LIN {X 0,Y 569.385,Z 629.743,A -85,B 0,C 180,E1 27677.459,E2 27677.459} C_VEL
LIN {X 0,Y 569.347,Z 629.746,A -85,B 0,C 180,E1 27674.085,E2 27674.085} C_VEL
LIN {X 0,Y 569.375,Z 629.741,A -85,B 0,C 180,E1 27670.786,E2 27670.786} C_VEL
LIN {X 0,Y 569.404,Z 629.994,A -85,B 0,C 180,E1 27669.564,E2 27669.564} C_VEL
LIN {X 0,Y 577.566,Z 654.883,A -85,B 0,C 180,E1 27666.47,E2 27666.47} C_VEL
LIN {X 0,Y 582.986,Z 672.69,A -85,B 0,C 180,E1 27664.382,E2 27664.382} C_VEL
LIN {X 0,Y 582.582,Z 679.276,A -85,B 0,C 180,E1 27663.798,E2 27663.798} C_VEL
LIN {X 0,Y 590.179,Z 717.868,A -85,B 0,C 180,E1 27662.715,E2 27662.715} C_VEL
LIN {X 0,Y 584.592,Z 960.2,A -85,B 0,C 180,E1 27659.286,E2 27659.286} C_VEL
LIN {X 0,Y 583.754,Z 989.804,A -85,B 0,C 180,E1 27658.818,E2 27658.818} C_VEL
LIN {X 0,Y 582.732,Z 1011.571,A -85,B 0,C 180,E1 27658.307,E2 27658.307} C_VEL
LIN {X 0,Y 581.47,Z 1033.5,A -85,B 0,C 180,E1 27657.607,E2 27657.607} C_VEL
LIN {X 0,Y 580.045,Z 1054.405,A -85,B 0,C 180,E1 27656.753,E2 27656.753} C_VEL
LIN {X 0,Y 578.394,Z 1076.21,A -85,B 0,C 180,E1 27655.657,E2 27655.657} C_VEL
LIN {X 0,Y 576.83,Z 1095.761,A -85,B 0,C 180,E1 27654.473,E2 27654.473} C_VEL
LIN {X 0,Y 575.231,Z 1114.452,A -85,B 0,C 180,E1 27653.13,E2 27653.13} C_VEL
LIN {X 0,Y 573.746,Z 1131.579,A -85,B 0,C 180,E1 27651.681,E2 27651.681} C_VEL
LIN {X 0,Y 572.318,Z 1148.38,A -85,B 0,C 180,E1 27650.023,E2 27650.023} C_VEL
LIN {X 0,Y 571.147,Z 1162.85,A -85,B 0,C 180,E1 27648.366,E2 27648.366} C_VEL
LIN {X 0,Y 570.1,Z 1176.631,A -85,B 0,C 180,E1 27646.505,E2 27646.505} C_VEL
LIN {X 0,Y 569.274,Z 1188.963,A -85,B 0,C 180,E1 27644.545,E2 27644.545} C_VEL
LIN {X 0,Y 568.7,Z 1199.347,A -85,B 0,C 180,E1 27642.591,E2 27642.591} C_VEL
LIN {X 0,Y 568.31,Z 1208.283,A -85,B 0,C 180,E1 27640.542,E2 27640.542} C_VEL
LIN {X 0,Y 568.098,Z 1215.604,A -85,B 0,C 180,E1 27638.439,E2 27638.439} C_VEL
LIN {X 0,Y 567.982,Z 1221.411,A -85,B 0,C 180,E1 27636.265,E2 27636.265} C_VEL
LIN {X 0,Y 567.957,Z 1225.194,A -85,B 0,C 180,E1 27634.239,E2 27634.239} C_VEL
LIN {X 0,Y 567.958,Z 1227.62,A -85,B 0,C 180,E1 27632.016,E2 27632.016} C_VEL
LIN {X 0,Y 567.959,Z 1228.354,A -85,B 0,C 180,E1 27629.898,E2 27629.898} C_VEL
LIN {X 0,Y 567.961,Z 1227.38,A -85,B 0,C 180,E1 27627.779,E2 27627.779} C_VEL
LIN {X 0,Y 567.963,Z 1224.652,A -85,B 0,C 180,E1 27625.556,E2 27625.556} C_VEL
LIN {X 0,Y 567.992,Z 1220.397,A -85,B 0,C 180,E1 27623.428,E2 27623.428} C_VEL
LIN {X 0,Y 568.113,Z 1214.604,A -85,B 0,C 180,E1 27621.395,E2 27621.395} C_VEL
LIN {X 0,Y 568.343,Z 1206.72,A -85,B 0,C 180,E1 27619.251,E2 27619.251} C_VEL
LIN {X 0,Y 568.733,Z 1197.343,A -85,B 0,C 180,E1 27617.2,E2 27617.2} C_VEL
LIN {X 0,Y 569.298,Z 1186.437,A -85,B 0,C 180,E1 27615.245,E2 27615.245} C_VEL
LIN {X 0,Y 570.048,Z 1174.137,A -85,B 0,C 180,E1 27613.386,E2 27613.386} C_VEL
LIN {X 0,Y 570.986,Z 1160.553,A -85,B 0,C 180,E1 27611.625,E2 27611.625} C_VEL
LIN {X 0,Y 572.146,Z 1144.814,A -85,B 0,C 180,E1 27609.89,E2 27609.89} C_VEL
LIN {X 0,Y 573.396,Z 1128.474,A -85,B 0,C 180,E1 27608.351,E2 27608.351} C_VEL
LIN {X 0,Y 574.818,Z 1109.922,A -85,B 0,C 180,E1 27606.85,E2 27606.85} C_VEL
LIN {X 0,Y 576.284,Z 1091.145,A -85,B 0,C 180,E1 27605.554,E2 27605.554} C_VEL
LIN {X 0,Y 577.77,Z 1070.527,A -85,B 0,C 180,E1 27604.363,E2 27604.363} C_VEL
LIN {X 0,Y 579.158,Z 1050.131,A -85,B 0,C 180,E1 27603.383,E2 27603.383} C_VEL
LIN {X 0,Y 580.584,Z 1027.426,A -85,B 0,C 180,E1 27602.493,E2 27602.493} C_VEL
LIN {X 0,Y 581.823,Z 1005.201,A -85,B 0,C 180,E1 27601.811,E2 27601.811} C_VEL
LIN {X 0,Y 582.893,Z 981.742,A -85,B 0,C 180,E1 27601.283,E2 27601.283} C_VEL
LIN {X 0,Y 586.569,Z 850.583,A -85,B 0,C 180,E1 27599.246,E2 27599.246} C_VEL
LIN {X 0,Y 590.83,Z 750.197,A -85,B 0,C 180,E1 27597.537,E2 27597.537} C_VEL
LIN {X 0,Y 592.379,Z 716.599,A -85,B 0,C 180,E1 27596.915,E2 27596.915} C_VEL
LIN {X 0,Y 588.657,Z 690.874,A -85,B 0,C 180,E1 27595.977,E2 27595.977} C_VEL
LIN {X 0,Y 585.547,Z 674.638,A -85,B 0,C 180,E1 27595.245,E2 27595.245} C_VEL
LIN {X 0,Y 583.11,Z 669.092,A -85,B 0,C 180,E1 27594.818,E2 27594.818} C_VEL
LIN {X 0,Y 580.106,Z 657.836,A -85,B 0,C 180,E1 27593.11,E2 27593.11} C_VEL
LIN {X 0,Y 577.035,Z 648.434,A -85,B 0,C 180,E1 27591.4,E2 27591.4} C_VEL
LIN {X 0,Y 574.123,Z 641.138,A -85,B 0,C 180,E1 27589.715,E2 27589.715} C_VEL
LIN {X 0,Y 572.591,Z 637.429,A -85,B 0,C 180,E1 27588.669,E2 27588.669} C_VEL
LIN {X 0,Y 570.972,Z 633.671,A -85,B 0,C 180,E1 27587.334,E2 27587.334} C_VEL
LIN {X 0,Y 569.377,Z 629.969,A -85,B 0,C 180,E1 27585.337,E2 27585.337} C_VEL
LIN {X 0,Y 569.384,Z 629.746,A -85,B 0,C 180,E1 27582.176,E2 27582.176} C_VEL
LIN {X 0,Y 569.39,Z 630.021,A -85,B 0,C 180,E1 27580.923,E2 27580.923} C_VEL
LIN {X 0,Y 571.02,Z 633.725,A -85,B 0,C 180,E1 27578.81,E2 27578.81} C_VEL
LIN {X 0,Y 573.022,Z 638.744,A -85,B 0,C 180,E1 27577.015,E2 27577.015} C_VEL
LIN {X 0,Y 574.473,Z 642.072,A -85,B 0,C 180,E1 27576.094,E2 27576.094} C_VEL
LIN {X 0,Y 579.186,Z 648.73,A -85,B 0,C 180,E1 27575.256,E2 27575.256} C_VEL
LIN {X 0,Y 583.805,Z 655.292,A -85,B 0,C 180,E1 27574.531,E2 27574.531} C_VEL
LIN {X 0,Y 590.369,Z 666.287,A -85,B 0,C 180,E1 27573.561,E2 27573.561} C_VEL
LIN {X 0,Y 594.016,Z 673.562,A -85,B 0,C 180,E1 27573.045,E2 27573.045} C_VEL
LIN {X 0,Y 588.975,Z 770.536,A -85,B 0,C 180,E1 27571.31,E2 27571.31} C_VEL
LIN {X 0,Y 585.467,Z 865.563,A -85,B 0,C 180,E1 27569.75,E2 27569.75} C_VEL
LIN {X 0,Y 583.506,Z 937.323,A -85,B 0,C 180,E1 27568.629,E2 27568.629} C_VEL
LIN {X 0,Y 582.639,Z 960.337,A -85,B 0,C 180,E1 27568.084,E2 27568.084} C_VEL
LIN {X 0,Y 581.532,Z 982.034,A -85,B 0,C 180,E1 27567.385,E2 27567.385} C_VEL
LIN {X 0,Y 580.245,Z 1003.436,A -85,B 0,C 180,E1 27566.509,E2 27566.509} C_VEL
LIN {X 0,Y 578.839,Z 1023.952,A -85,B 0,C 180,E1 27565.477,E2 27565.477} C_VEL
LIN {X 0,Y 577.353,Z 1043.592,A -85,B 0,C 180,E1 27564.289,E2 27564.289} C_VEL
LIN {X 0,Y 575.82,Z 1062.116,A -85,B 0,C 180,E1 27562.946,E2 27562.946} C_VEL
LIN {X 0,Y 574.347,Z 1079.125,A -85,B 0,C 180,E1 27561.495,E2 27561.495} C_VEL
LIN {X 0,Y 572.947,Z 1095.168,A -85,B 0,C 180,E1 27559.897,E2 27559.897} C_VEL
LIN {X 0,Y 571.741,Z 1109.387,A -85,B 0,C 180,E1 27558.245,E2 27558.245} C_VEL
LIN {X 0,Y 570.667,Z 1122.187,A -85,B 0,C 180,E1 27556.492,E2 27556.492} C_VEL
LIN {X 0,Y 569.736,Z 1134.33,A -85,B 0,C 180,E1 27554.537,E2 27554.537} C_VEL
LIN {X 0,Y 569.076,Z 1144.509,A -85,B 0,C 180,E1 27552.586,E2 27552.586} C_VEL
LIN {X 0,Y 568.574,Z 1153.183,A -85,B 0,C 180,E1 27550.54,E2 27550.54} C_VEL
LIN {X 0,Y 568.254,Z 1160.43,A -85,B 0,C 180,E1 27548.4,E2 27548.4} C_VEL
LIN {X 0,Y 568.086,Z 1165.74,A -85,B 0,C 180,E1 27546.368,E2 27546.368} C_VEL
LIN {X 0,Y 567.995,Z 1169.579,A -85,B 0,C 180,E1 27544.242,E2 27544.242} C_VEL
LIN {X 0,Y 567.96,Z 1171.94,A -85,B 0,C 180,E1 27542.02,E2 27542.02} C_VEL
LIN {X 0,Y 567.963,Z 1172.683,A -85,B 0,C 180,E1 27539.901,E2 27539.901} C_VEL
LIN {X 0,Y 567.956,Z 1171.775,A -85,B 0,C 180,E1 27537.783,E2 27537.783} C_VEL
LIN {X 0,Y 567.991,Z 1169.228,A -85,B 0,C 180,E1 27535.56,E2 27535.56} C_VEL
LIN {X 0,Y 568.078,Z 1165.231,A -85,B 0,C 180,E1 27533.433,E2 27533.433} C_VEL
LIN {X 0,Y 568.246,Z 1159.452,A -85,B 0,C 180,E1 27531.299,E2 27531.299} C_VEL
LIN {X 0,Y 568.575,Z 1151.939,A -85,B 0,C 180,E1 27529.157,E2 27529.157} C_VEL
LIN {X 0,Y 569.088,Z 1143.026,A -85,B 0,C 180,E1 27527.109,E2 27527.109} C_VEL
LIN {X 0,Y 569.782,Z 1132.656,A -85,B 0,C 180,E1 27525.157,E2 27525.157} C_VEL
LIN {X 0,Y 570.734,Z 1120.273,A -85,B 0,C 180,E1 27523.2,E2 27523.2} C_VEL
LIN {X 0,Y 571.903,Z 1106.402,A -85,B 0,C 180,E1 27521.343,E2 27521.343} C_VEL
LIN {X 0,Y 573.241,Z 1091.506,A -85,B 0,C 180,E1 27519.639,E2 27519.639} C_VEL
LIN {X 0,Y 574.707,Z 1074.964,A -85,B 0,C 180,E1 27518.036,E2 27518.036} C_VEL
LIN {X 0,Y 576.258,Z 1057.5,A -85,B 0,C 180,E1 27516.59,E2 27516.59} C_VEL
LIN {X 0,Y 577.834,Z 1039.197,A -85,B 0,C 180,E1 27515.295,E2 27515.295} C_VEL
LIN {X 0,Y 579.41,Z 1019.369,A -85,B 0,C 180,E1 27514.116,E2 27514.116} C_VEL
LIN {X 0,Y 580.837,Z 999.457,A -85,B 0,C 180,E1 27513.138,E2 27513.138} C_VEL
LIN {X 0,Y 582.221,Z 977.603,A -85,B 0,C 180,E1 27512.266,E2 27512.266} C_VEL
LIN {X 0,Y 583.325,Z 956.104,A -85,B 0,C 180,E1 27511.593,E2 27511.593} C_VEL
LIN {X 0,Y 584.219,Z 933.964,A -85,B 0,C 180,E1 27511.089,E2 27511.089} C_VEL
LIN {X 0,Y 585.088,Z 897.354,A -85,B 0,C 180,E1 27510.542,E2 27510.542} C_VEL
LIN {X 0,Y 590.004,Z 687.581,A -85,B 0,C 180,E1 27507.575,E2 27507.575} C_VEL
LIN {X 0,Y 590.303,Z 670.134,A -85,B 0,C 180,E1 27507.312,E2 27507.312} C_VEL
LIN {X 0,Y 576.833,Z 644.025,A -85,B 0,C 180,E1 27506.064,E2 27506.064} C_VEL
LIN {X 0,Y 569.547,Z 630.919,A -85,B 0,C 180,E1 27505.383,E2 27505.383} C_VEL
LIN {X 0,Y 569.316,Z 629.751,A -85,B 0,C 180,E1 27505.32,E2 27505.32} C_VEL
LIN {X 0,Y 569.345,Z 629.744,A -85,B 0,C 180,E1 27501.948,E2 27501.948} C_VEL
LIN {X 0,Y 569.377,Z 629.741,A -85,B 0,C 180,E1 27498.732,E2 27498.732} C_VEL
LIN {X 0,Y 569.363,Z 629.745,A -85,B 0,C 180,E1 27496.965,E2 27496.965} C_VEL
LIN {X 0,Y 568.378,Z 629.865,A -85,B 0,C 180,E1 27496.19,E2 27496.19} C_VEL
LIN {X 0,Y 561.876,Z 630.685,A -85,B 0,C 180,E1 27493.958,E2 27493.958} C_VEL
LIN {X 0,Y 561.411,Z 630.738,A -85,B 0,C 180,E1 27493.448,E2 27493.448} C_VEL
LIN {X 0,Y 561.412,Z 630.736,A -85,B 0,C 180,E1 27490.28,E2 27490.28} C_VEL
LIN {X 0,Y 561.376,Z 630.737,A -85,B 0,C 180,E1 27487.016,E2 27487.016} C_VEL
LIN {X 0,Y 561.425,Z 630.732,A -85,B 0,C 180,E1 27483.73,E2 27483.73} C_VEL
LIN {X 0,Y 561.432,Z 630.733,A -85,B 0,C 180,E1 27480.466,E2 27480.466} C_VEL
LIN {X 0,Y 561.439,Z 630.736,A -85,B 0,C 180,E1 27477.125,E2 27477.125} C_VEL
LIN {X 0,Y 561.416,Z 630.737,A -85,B 0,C 180,E1 27473.848,E2 27473.848} C_VEL
LIN {X 0,Y 561.36,Z 630.74,A -85,B 0,C 180,E1 27470.652,E2 27470.652} C_VEL
LIN {X 0,Y 561.43,Z 630.731,A -85,B 0,C 180,E1 27467.411,E2 27467.411} C_VEL
LIN {X 0,Y 561.446,Z 630.727,A -85,B 0,C 180,E1 27464.123,E2 27464.123} C_VEL
LIN {X 0,Y 561.438,Z 630.735,A -85,B 0,C 180,E1 27460.675,E2 27460.675} C_VEL
LIN {X 0,Y 561.421,Z 630.727,A -85,B 0,C 180,E1 27457.369,E2 27457.369} C_VEL
LIN {X 0,Y 561.36,Z 630.737,A -85,B 0,C 180,E1 27454.127,E2 27454.127} C_VEL
LIN {X 0,Y 561.413,Z 630.734,A -85,B 0,C 180,E1 27450.818,E2 27450.818} C_VEL
LIN {X 0,Y 561.429,Z 630.732,A -85,B 0,C 180,E1 27447.654,E2 27447.654} C_VEL
LIN {X 0,Y 561.43,Z 630.727,A -85,B 0,C 180,E1 27444.278,E2 27444.278} C_VEL
LIN {X 0,Y 561.417,Z 630.729,A -85,B 0,C 180,E1 27441.088,E2 27441.088} C_VEL
LIN {X 0,Y 561.379,Z 630.731,A -85,B 0,C 180,E1 27437.765,E2 27437.765} C_VEL
LIN {X 0,Y 561.424,Z 630.736,A -85,B 0,C 180,E1 27434.507,E2 27434.507} C_VEL
LIN {X 0,Y 561.404,Z 630.736,A -85,B 0,C 180,E1 27431.303,E2 27431.303} C_VEL
LIN {X 0,Y 561.42,Z 630.732,A -85,B 0,C 180,E1 27427.929,E2 27427.929} C_VEL
LIN {X 0,Y 561.423,Z 630.731,A -85,B 0,C 180,E1 27424.697,E2 27424.697} C_VEL
LIN {X 0,Y 561.402,Z 630.738,A -85,B 0,C 180,E1 27421.375,E2 27421.375} C_VEL
LIN {X 0,Y 561.422,Z 630.739,A -85,B 0,C 180,E1 27418.188,E2 27418.188} C_VEL
LIN {X 0,Y 561.378,Z 630.739,A -85,B 0,C 180,E1 27415.006,E2 27415.006} C_VEL
LIN {X 0,Y 561.423,Z 630.732,A -85,B 0,C 180,E1 27411.702,E2 27411.702} C_VEL
LIN {X 0,Y 561.433,Z 630.734,A -85,B 0,C 180,E1 27408.413,E2 27408.413} C_VEL
LIN {X 0,Y 561.427,Z 630.732,A -85,B 0,C 180,E1 27405.008,E2 27405.008} C_VEL
LIN {X 0,Y 561.397,Z 630.839,A -85,B 0,C 180,E1 27402.628,E2 27402.628} C_VEL
LIN {X 0,Y 569.252,Z 659.307,A -85,B 0,C 180,E1 27400.003,E2 27400.003} C_VEL
LIN {X 0,Y 568.967,Z 679.663,A -85,B 0,C 180,E1 27398.395,E2 27398.395} C_VEL
LIN {X 0,Y 568.05,Z 720.365,A -85,B 0,C 180,E1 27395.199,E2 27395.199} C_VEL
LIN {X 0,Y 567.025,Z 761.508,A -85,B 0,C 180,E1 27391.988,E2 27391.988} C_VEL
LIN {X 0,Y 565.993,Z 804.914,A -85,B 0,C 180,E1 27388.601,E2 27388.601} C_VEL
LIN {X 0,Y 565.449,Z 830.086,A -85,B 0,C 180,E1 27386.664,E2 27386.664} C_VEL
LIN {X 0,Y 565.724,Z 838.01,A -85,B 0,C 180,E1 27386.539,E2 27386.539} C_VEL
LIN {X 0,Y 564.249,Z 973.158,A -85,B 0,C 180,E1 27384.603,E2 27384.603} C_VEL
LIN {X 0,Y 564.09,Z 989.543,A -85,B 0,C 180,E1 27384.179,E2 27384.179} C_VEL
LIN {X 0,Y 563.794,Z 1005.741,A -85,B 0,C 180,E1 27383.565,E2 27383.565} C_VEL
LIN {X 0,Y 563.396,Z 1021.256,A -85,B 0,C 180,E1 27382.759,E2 27382.759} C_VEL
LIN {X 0,Y 562.976,Z 1035.029,A -85,B 0,C 180,E1 27381.842,E2 27381.842} C_VEL
LIN {X 0,Y 562.482,Z 1048.394,A -85,B 0,C 180,E1 27380.714,E2 27380.714} C_VEL
LIN {X 0,Y 562.053,Z 1059.619,A -85,B 0,C 180,E1 27379.536,E2 27379.536} C_VEL
LIN {X 0,Y 561.626,Z 1070.156,A -85,B 0,C 180,E1 27378.151,E2 27378.151} C_VEL
LIN {X 0,Y 561.317,Z 1078.466,A -85,B 0,C 180,E1 27376.77,E2 27376.77} C_VEL
LIN {X 0,Y 561.071,Z 1085.768,A -85,B 0,C 180,E1 27375.184,E2 27375.184} C_VEL
LIN {X 0,Y 560.935,Z 1090.731,A -85,B 0,C 180,E1 27373.712,E2 27373.712} C_VEL
LIN {X 0,Y 560.847,Z 1094.409,A -85,B 0,C 180,E1 27372.037,E2 27372.037} C_VEL
LIN {X 0,Y 560.842,Z 1096.156,A -85,B 0,C 180,E1 27370.475,E2 27370.475} C_VEL
LIN {X 0,Y 560.902,Z 1096.156,A -85,B 0,C 180,E1 27368.816,E2 27368.816} C_VEL
LIN {X 0,Y 561.028,Z 1094.371,A -85,B 0,C 180,E1 27367.164,E2 27367.164} C_VEL
LIN {X 0,Y 561.233,Z 1090.637,A -85,B 0,C 180,E1 27365.518,E2 27365.518} C_VEL
LIN {X 0,Y 561.523,Z 1085.354,A -85,B 0,C 180,E1 27363.98,E2 27363.98} C_VEL
LIN {X 0,Y 561.906,Z 1078.031,A -85,B 0,C 180,E1 27362.445,E2 27362.445} C_VEL
LIN {X 0,Y 562.345,Z 1069.862,A -85,B 0,C 180,E1 27361.118,E2 27361.118} C_VEL
LIN {X 0,Y 562.879,Z 1059.478,A -85,B 0,C 180,E1 27359.794,E2 27359.794} C_VEL
LIN {X 0,Y 563.425,Z 1048.063,A -85,B 0,C 180,E1 27358.625,E2 27358.625} C_VEL
LIN {X 0,Y 563.966,Z 1034.953,A -85,B 0,C 180,E1 27357.559,E2 27357.559} C_VEL
LIN {X 0,Y 564.394,Z 1021.683,A -85,B 0,C 180,E1 27356.697,E2 27356.697} C_VEL
LIN {X 0,Y 564.758,Z 1007.443,A -85,B 0,C 180,E1 27355.988,E2 27355.988} C_VEL
LIN {X 0,Y 565.014,Z 993.479,A -85,B 0,C 180,E1 27355.462,E2 27355.462} C_VEL
LIN {X 0,Y 565.148,Z 978.324,A -85,B 0,C 180,E1 27355.047,E2 27355.047} C_VEL
LIN {X 0,Y 565.439,Z 937.108,A -85,B 0,C 180,E1 27354.417,E2 27354.417} C_VEL
LIN {X 0,Y 567.178,Z 836.214,A -85,B 0,C 180,E1 27352.884,E2 27352.884} C_VEL
LIN {X 0,Y 568.054,Z 809.4,A -85,B 0,C 180,E1 27350.832,E2 27350.832} C_VEL
LIN {X 0,Y 568.945,Z 767.932,A -85,B 0,C 180,E1 27347.669,E2 27347.669} C_VEL
LIN {X 0,Y 569.778,Z 726.71,A -85,B 0,C 180,E1 27344.58,E2 27344.58} C_VEL
LIN {X 0,Y 570.332,Z 682.729,A -85,B 0,C 180,E1 27341.338,E2 27341.338} C_VEL
LIN {X 0,Y 570.591,Z 658.561,A -85,B 0,C 180,E1 27339.589,E2 27339.589} C_VEL
LIN {X 0,Y 565.651,Z 642.355,A -85,B 0,C 180,E1 27338.099,E2 27338.099} C_VEL
LIN {X 0,Y 561.428,Z 630.743,A -85,B 0,C 180,E1 27336.961,E2 27336.961} C_VEL
LIN {X 0,Y 561.44,Z 630.737,A -85,B 0,C 180,E1 27333.446,E2 27333.446} C_VEL
LIN {X 0,Y 561.448,Z 630.735,A -85,B 0,C 180,E1 27330.087,E2 27330.087} C_VEL
LIN {X 0,Y 561.403,Z 630.738,A -85,B 0,C 180,E1 27326.645,E2 27326.645} C_VEL
LIN {X 0,Y 561.437,Z 630.734,A -85,B 0,C 180,E1 27323.37,E2 27323.37} C_VEL
LIN {X 0,Y 561.423,Z 630.736,A -85,B 0,C 180,E1 27320.12,E2 27320.12} C_VEL
LIN {X 0,Y 561.434,Z 630.731,A -85,B 0,C 180,E1 27316.602,E2 27316.602} C_VEL
LIN {X 0,Y 561.444,Z 630.732,A -85,B 0,C 180,E1 27313.246,E2 27313.246} C_VEL
LIN {X 0,Y 561.42,Z 630.863,A -85,B 0,C 180,E1 27310.044,E2 27310.044} C_VEL
LIN {X 0,Y 569.404,Z 655.178,A -85,B 0,C 180,E1 27306.964,E2 27306.964} C_VEL
LIN {X 0,Y 575.608,Z 675.318,A -85,B 0,C 180,E1 27304.573,E2 27304.573} C_VEL
LIN {X 0,Y 575.395,Z 678.971,A -85,B 0,C 180,E1 27304.253,E2 27304.253} C_VEL
LIN {X 0,Y 583.269,Z 719.277,A -85,B 0,C 180,E1 27303.096,E2 27303.096} C_VEL
LIN {X 0,Y 577.417,Z 957.319,A -85,B 0,C 180,E1 27299.665,E2 27299.665} C_VEL
LIN {X 0,Y 576.498,Z 989.006,A -85,B 0,C 180,E1 27299.162,E2 27299.162} C_VEL
LIN {X 0,Y 575.424,Z 1011.077,A -85,B 0,C 180,E1 27298.639,E2 27298.639} C_VEL
LIN {X 0,Y 574.102,Z 1032.922,A -85,B 0,C 180,E1 27297.935,E2 27297.935} C_VEL
LIN {X 0,Y 572.631,Z 1053.761,A -85,B 0,C 180,E1 27297.079,E2 27297.079} C_VEL
LIN {X 0,Y 570.975,Z 1074.812,A -85,B 0,C 180,E1 27296.017,E2 27296.017} C_VEL
LIN {X 0,Y 569.331,Z 1094.614,A -85,B 0,C 180,E1 27294.816,E2 27294.816} C_VEL
LIN {X 0,Y 567.639,Z 1113.377,A -85,B 0,C 180,E1 27293.457,E2 27293.457} C_VEL
LIN {X 0,Y 566.07,Z 1130.813,A -85,B 0,C 180,E1 27291.973,E2 27291.973} C_VEL
LIN {X 0,Y 564.573,Z 1147.561,A -85,B 0,C 180,E1 27290.31,E2 27290.31} C_VEL
LIN {X 0,Y 563.301,Z 1162.551,A -85,B 0,C 180,E1 27288.577,E2 27288.577} C_VEL
LIN {X 0,Y 562.228,Z 1175.993,A -85,B 0,C 180,E1 27286.743,E2 27286.743} C_VEL
LIN {X 0,Y 561.357,Z 1188.387,A -85,B 0,C 180,E1 27284.755,E2 27284.755} C_VEL
LIN {X 0,Y 560.738,Z 1199.01,A -85,B 0,C 180,E1 27282.733,E2 27282.733} C_VEL
LIN {X 0,Y 560.336,Z 1207.801,A -85,B 0,C 180,E1 27280.693,E2 27280.693} C_VEL
LIN {X 0,Y 560.108,Z 1214.976,A -85,B 0,C 180,E1 27278.623,E2 27278.623} C_VEL
LIN {X 0,Y 559.987,Z 1220.791,A -85,B 0,C 180,E1 27276.457,E2 27276.457} C_VEL
LIN {X 0,Y 559.962,Z 1224.633,A -85,B 0,C 180,E1 27274.402,E2 27274.402} C_VEL
LIN {X 0,Y 559.966,Z 1227.162,A -85,B 0,C 180,E1 27272.148,E2 27272.148} C_VEL
LIN {X 0,Y 559.979,Z 1227.98,A -85,B 0,C 180,E1 27269.999,E2 27269.999} C_VEL
LIN {X 0,Y 559.971,Z 1227.048,A -85,B 0,C 180,E1 27267.85,E2 27267.85} C_VEL
LIN {X 0,Y 559.97,Z 1224.389,A -85,B 0,C 180,E1 27265.595,E2 27265.595} C_VEL
LIN {X 0,Y 559.995,Z 1220.181,A -85,B 0,C 180,E1 27263.437,E2 27263.437} C_VEL
LIN {X 0,Y 560.114,Z 1214.408,A -85,B 0,C 180,E1 27261.375,E2 27261.375} C_VEL
LIN {X 0,Y 560.35,Z 1206.582,A -85,B 0,C 180,E1 27259.2,E2 27259.2} C_VEL
LIN {X 0,Y 560.753,Z 1197.256,A -85,B 0,C 180,E1 27257.12,E2 27257.12} C_VEL
LIN {X 0,Y 561.339,Z 1186.369,A -85,B 0,C 180,E1 27255.136,E2 27255.136} C_VEL
LIN {X 0,Y 562.121,Z 1174.12,A -85,B 0,C 180,E1 27253.251,E2 27253.251} C_VEL
LIN {X 0,Y 563.103,Z 1160.613,A -85,B 0,C 180,E1 27251.466,E2 27251.466} C_VEL
LIN {X 0,Y 564.333,Z 1144.635,A -85,B 0,C 180,E1 27249.678,E2 27249.678} C_VEL
LIN {X 0,Y 565.671,Z 1128.13,A -85,B 0,C 180,E1 27248.1,E2 27248.1} C_VEL
LIN {X 0,Y 567.119,Z 1110.25,A -85,B 0,C 180,E1 27246.627,E2 27246.627} C_VEL
LIN {X 0,Y 568.715,Z 1090.798,A -85,B 0,C 180,E1 27245.263,E2 27245.263} C_VEL
LIN {X 0,Y 570.288,Z 1070.235,A -85,B 0,C 180,E1 27244.058,E2 27244.058} C_VEL
LIN {X 0,Y 571.75,Z 1049.961,A -85,B 0,C 180,E1 27243.066,E2 27243.066} C_VEL
LIN {X 0,Y 573.258,Z 1027.548,A -85,B 0,C 180,E1 27242.17,E2 27242.17} C_VEL
LIN {X 0,Y 574.603,Z 1005.011,A -85,B 0,C 180,E1 27241.462,E2 27241.462} C_VEL
LIN {X 0,Y 575.773,Z 981.249,A -85,B 0,C 180,E1 27240.915,E2 27240.915} C_VEL
LIN {X 0,Y 579.704,Z 854.385,A -85,B 0,C 180,E1 27238.881,E2 27238.881} C_VEL
LIN {X 0,Y 584.375,Z 753.94,A -85,B 0,C 180,E1 27237.115,E2 27237.115} C_VEL
LIN {X 0,Y 586.236,Z 718.159,A -85,B 0,C 180,E1 27236.433,E2 27236.433} C_VEL
LIN {X 0,Y 582.964,Z 693.73,A -85,B 0,C 180,E1 27235.504,E2 27235.504} C_VEL
LIN {X 0,Y 580.226,Z 678.94,A -85,B 0,C 180,E1 27234.818,E2 27234.818} C_VEL
LIN {X 0,Y 576.409,Z 670.73,A -85,B 0,C 180,E1 27234.129,E2 27234.129} C_VEL
LIN {X 0,Y 575.133,Z 667.897,A -85,B 0,C 180,E1 27233.887,E2 27233.887} C_VEL
LIN {X 0,Y 572.098,Z 657.429,A -85,B 0,C 180,E1 27232.105,E2 27232.105} C_VEL
LIN {X 0,Y 569.328,Z 649.511,A -85,B 0,C 180,E1 27230.446,E2 27230.446} C_VEL
LIN {X 0,Y 567.055,Z 643.417,A -85,B 0,C 180,E1 27228.847,E2 27228.847} C_VEL
LIN {X 0,Y 565.079,Z 639.052,A -85,B 0,C 180,E1 27227.252,E2 27227.252} C_VEL
LIN {X 0,Y 563.608,Z 635.39,A -85,B 0,C 180,E1 27225.207,E2 27225.207} C_VEL
LIN {X 0,Y 562.847,Z 634.42,A -85,B 0,C 180,E1 27223.25,E2 27223.25} C_VEL
LIN {X 0,Y 563.487,Z 635.206,A -85,B 0,C 180,E1 27221.203,E2 27221.203} C_VEL
LIN {X 0,Y 564.786,Z 638.691,A -85,B 0,C 180,E1 27219.071,E2 27219.071} C_VEL
LIN {X 0,Y 565.483,Z 640.302,A -85,B 0,C 180,E1 27218.365,E2 27218.365} C_VEL
LIN {X 0,Y 566.994,Z 643.842,A -85,B 0,C 180,E1 27217.145,E2 27217.145} C_VEL
LIN {X 0,Y 571.237,Z 649.469,A -85,B 0,C 180,E1 27216.275,E2 27216.275} C_VEL
LIN {X 0,Y 577.123,Z 657.628,A -85,B 0,C 180,E1 27215.224,E2 27215.224} C_VEL
LIN {X 0,Y 584.224,Z 669.254,A -85,B 0,C 180,E1 27214.091,E2 27214.091} C_VEL
LIN {X 0,Y 587.987,Z 676.825,A -85,B 0,C 180,E1 27213.519,E2 27213.519} C_VEL
LIN {X 0,Y 582.457,Z 772.876,A -85,B 0,C 180,E1 27211.741,E2 27211.741} C_VEL
LIN {X 0,Y 578.648,Z 865.794,A -85,B 0,C 180,E1 27210.161,E2 27210.161} C_VEL
LIN {X 0,Y 576.432,Z 938.317,A -85,B 0,C 180,E1 27208.989,E2 27208.989} C_VEL
LIN {X 0,Y 575.504,Z 961.305,A -85,B 0,C 180,E1 27208.43,E2 27208.43} C_VEL
LIN {X 0,Y 574.344,Z 982.62,A -85,B 0,C 180,E1 27207.729,E2 27207.729} C_VEL
LIN {X 0,Y 573.023,Z 1003.357,A -85,B 0,C 180,E1 27206.87,E2 27206.87} C_VEL
LIN {X 0,Y 571.616,Z 1023.035,A -85,B 0,C 180,E1 27205.878,E2 27205.878} C_VEL
LIN {X 0,Y 570.033,Z 1042.814,A -85,B 0,C 180,E1 27204.677,E2 27204.677} C_VEL
LIN {X 0,Y 568.421,Z 1061.346,A -85,B 0,C 180,E1 27203.33,E2 27203.33} C_VEL
LIN {X 0,Y 566.842,Z 1078.642,A -85,B 0,C 180,E1 27201.853,E2 27201.853} C_VEL
LIN {X 0,Y 565.41,Z 1094.414,A -85,B 0,C 180,E1 27200.282,E2 27200.282} C_VEL
LIN {X 0,Y 564.094,Z 1108.738,A -85,B 0,C 180,E1 27198.608,E2 27198.608} C_VEL
LIN {X 0,Y 562.914,Z 1122.075,A -85,B 0,C 180,E1 27196.78,E2 27196.78} C_VEL
LIN {X 0,Y 561.942,Z 1134.049,A -85,B 0,C 180,E1 27194.848,E2 27194.848} C_VEL
LIN {X 0,Y 561.215,Z 1144.327,A -85,B 0,C 180,E1 27192.87,E2 27192.87} C_VEL
LIN {X 0,Y 560.659,Z 1153.124,A -85,B 0,C 180,E1 27190.795,E2 27190.795} C_VEL
LIN {X 0,Y 560.301,Z 1160.499,A -85,B 0,C 180,E1 27188.623,E2 27188.623} C_VEL
LIN {X 0,Y 560.117,Z 1165.903,A -85,B 0,C 180,E1 27186.562,E2 27186.562} C_VEL
LIN {X 0,Y 560.016,Z 1169.818,A -85,B 0,C 180,E1 27184.405,E2 27184.405} C_VEL
LIN {X 0,Y 559.97,Z 1172.274,A -85,B 0,C 180,E1 27182.151,E2 27182.151} C_VEL
LIN {X 0,Y 559.976,Z 1173.077,A -85,B 0,C 180,E1 27180.002,E2 27180.002} C_VEL
LIN {X 0,Y 559.967,Z 1172.223,A -85,B 0,C 180,E1 27177.853,E2 27177.853} C_VEL
LIN {X 0,Y 560.001,Z 1169.739,A -85,B 0,C 180,E1 27175.599,E2 27175.599} C_VEL
LIN {X 0,Y 560.093,Z 1165.774,A -85,B 0,C 180,E1 27173.442,E2 27173.442} C_VEL
LIN {X 0,Y 560.271,Z 1160.043,A -85,B 0,C 180,E1 27171.277,E2 27171.277} C_VEL
LIN {X 0,Y 560.617,Z 1152.578,A -85,B 0,C 180,E1 27169.105,E2 27169.105} C_VEL
LIN {X 0,Y 561.155,Z 1143.71,A -85,B 0,C 180,E1 27167.028,E2 27167.028} C_VEL
LIN {X 0,Y 561.88,Z 1133.353,A -85,B 0,C 180,E1 27165.049,E2 27165.049} C_VEL
LIN {X 0,Y 562.876,Z 1121.016,A -85,B 0,C 180,E1 27163.065,E2 27163.065} C_VEL
LIN {X 0,Y 564.025,Z 1108.041,A -85,B 0,C 180,E1 27161.287,E2 27161.287} C_VEL
LIN {X 0,Y 565.345,Z 1093.701,A -85,B 0,C 180,E1 27159.612,E2 27159.612} C_VEL
LIN {X 0,Y 566.85,Z 1077.501,A -85,B 0,C 180,E1 27157.989,E2 27157.989} C_VEL
LIN {X 0,Y 568.514,Z 1059.793,A -85,B 0,C 180,E1 27156.472,E2 27156.472} C_VEL
LIN {X 0,Y 570.196,Z 1041.149,A -85,B 0,C 180,E1 27155.114,E2 27155.114} C_VEL
LIN {X 0,Y 571.828,Z 1021.367,A -85,B 0,C 180,E1 27153.914,E2 27153.914} C_VEL
LIN {X 0,Y 573.384,Z 1000.703,A -85,B 0,C 180,E1 27152.873,E2 27152.873} C_VEL
LIN {X 0,Y 574.821,Z 979.108,A -85,B 0,C 180,E1 27151.991,E2 27151.991} C_VEL
LIN {X 0,Y 576.001,Z 957.331,A -85,B 0,C 180,E1 27151.291,E2 27151.291} C_VEL
LIN {X 0,Y 576.942,Z 934.879,A -85,B 0,C 180,E1 27150.769,E2 27150.769} C_VEL
LIN {X 0,Y 577.783,Z 902.166,A -85,B 0,C 180,E1 27150.265,E2 27150.265} C_VEL
LIN {X 0,Y 582.919,Z 694.857,A -85,B 0,C 180,E1 27147.281,E2 27147.281} C_VEL
LIN {X 0,Y 583.379,Z 672.772,A -85,B 0,C 180,E1 27146.944,E2 27146.944} C_VEL
LIN {X 0,Y 570.933,Z 648.601,A -85,B 0,C 180,E1 27145.777,E2 27145.777} C_VEL
LIN {X 0,Y 561.672,Z 631.972,A -85,B 0,C 180,E1 27144.886,E2 27144.886} C_VEL
LIN {X 0,Y 561.424,Z 630.735,A -85,B 0,C 180,E1 27144.834,E2 27144.834} C_VEL
LIN {X 0,Y 561.408,Z 630.734,A -85,B 0,C 180,E1 27141.572,E2 27141.572} C_VEL
LIN {X 0,Y 561.44,Z 630.727,A -85,B 0,C 180,E1 27138.24,E2 27138.24} C_VEL
LIN {X 0,Y 561.409,Z 630.734,A -85,B 0,C 180,E1 27134.998,E2 27134.998} C_VEL
LIN {X 0,Y 561.411,Z 630.738,A -85,B 0,C 180,E1 27133.448,E2 27133.448} C_VEL
LIN {X 0,Y 560.405,Z 630.86,A -85,B 0,C 180,E1 27132.662,E2 27132.662} C_VEL
LIN {X 0,Y 553.949,Z 631.666,A -85,B 0,C 180,E1 27130.398,E2 27130.398} C_VEL
LIN {X 0,Y 553.472,Z 631.726,A -85,B 0,C 180,E1 27129.881,E2 27129.881} C_VEL
LIN {X 0,Y 553.457,Z 631.727,A -85,B 0,C 180,E1 27126.67,E2 27126.67} C_VEL
LIN {X 0,Y 553.471,Z 631.723,A -85,B 0,C 180,E1 27123.313,E2 27123.313} C_VEL
LIN {X 0,Y 553.5,Z 631.718,A -85,B 0,C 180,E1 27120.027,E2 27120.027} C_VEL
LIN {X 0,Y 553.468,Z 631.722,A -85,B 0,C 180,E1 27116.619,E2 27116.619} C_VEL
LIN {X 0,Y 553.477,Z 631.725,A -85,B 0,C 180,E1 27113.307,E2 27113.307} C_VEL
LIN {X 0,Y 553.451,Z 631.729,A -85,B 0,C 180,E1 27110.05,E2 27110.05} C_VEL
LIN {X 0,Y 553.459,Z 631.722,A -85,B 0,C 180,E1 27106.774,E2 27106.774} C_VEL
LIN {X 0,Y 553.502,Z 631.711,A -85,B 0,C 180,E1 27103.477,E2 27103.477} C_VEL
LIN {X 0,Y 553.478,Z 631.721,A -85,B 0,C 180,E1 27100.094,E2 27100.094} C_VEL
LIN {X 0,Y 553.488,Z 631.724,A -85,B 0,C 180,E1 27096.745,E2 27096.745} C_VEL
LIN {X 0,Y 553.442,Z 631.726,A -85,B 0,C 180,E1 27093.523,E2 27093.523} C_VEL
LIN {X 0,Y 553.443,Z 631.724,A -85,B 0,C 180,E1 27090.208,E2 27090.208} C_VEL
LIN {X 0,Y 553.5,Z 631.71,A -85,B 0,C 180,E1 27086.998,E2 27086.998} C_VEL
LIN {X 0,Y 553.489,Z 631.723,A -85,B 0,C 180,E1 27083.571,E2 27083.571} C_VEL
LIN {X 0,Y 553.497,Z 631.716,A -85,B 0,C 180,E1 27080.225,E2 27080.225} C_VEL
LIN {X 0,Y 553.456,Z 631.718,A -85,B 0,C 180,E1 27076.95,E2 27076.95} C_VEL
LIN {X 0,Y 553.43,Z 631.725,A -85,B 0,C 180,E1 27073.631,E2 27073.631} C_VEL
LIN {X 0,Y 553.494,Z 631.718,A -85,B 0,C 180,E1 27070.368,E2 27070.368} C_VEL
LIN {X 0,Y 553.499,Z 631.721,A -85,B 0,C 180,E1 27067.035,E2 27067.035} C_VEL
LIN {X 0,Y 553.501,Z 631.723,A -85,B 0,C 180,E1 27063.617,E2 27063.617} C_VEL
LIN {X 0,Y 553.483,Z 631.723,A -85,B 0,C 180,E1 27060.33,E2 27060.33} C_VEL
LIN {X 0,Y 553.423,Z 631.729,A -85,B 0,C 180,E1 27057.058,E2 27057.058} C_VEL
LIN {X 0,Y 553.48,Z 631.723,A -85,B 0,C 180,E1 27053.793,E2 27053.793} C_VEL
LIN {X 0,Y 553.503,Z 631.723,A -85,B 0,C 180,E1 27050.472,E2 27050.472} C_VEL
LIN {X 0,Y 553.501,Z 631.72,A -85,B 0,C 180,E1 27047.078,E2 27047.078} C_VEL
LIN {X 0,Y 553.498,Z 631.722,A -85,B 0,C 180,E1 27043.734,E2 27043.734} C_VEL
LIN {X 0,Y 553.489,Z 631.938,A -85,B 0,C 180,E1 27042.922,E2 27042.922} C_VEL
LIN {X 0,Y 560.925,Z 658.539,A -85,B 0,C 180,E1 27040.437,E2 27040.437} C_VEL
LIN {X 0,Y 561.87,Z 662.932,A -85,B 0,C 180,E1 27040.042,E2 27040.042} C_VEL
LIN {X 0,Y 560.796,Z 706.476,A -85,B 0,C 180,E1 27036.609,E2 27036.609} C_VEL
LIN {X 0,Y 559.746,Z 748.66,A -85,B 0,C 180,E1 27033.284,E2 27033.284} C_VEL
LIN {X 0,Y 558.651,Z 789.577,A -85,B 0,C 180,E1 27030.073,E2 27030.073} C_VEL
LIN {X 0,Y 557.718,Z 830.829,A -85,B 0,C 180,E1 27026.865,E2 27026.865} C_VEL
LIN {X 0,Y 557.977,Z 839.074,A -85,B 0,C 180,E1 27026.734,E2 27026.734} C_VEL
LIN {X 0,Y 556.415,Z 973.992,A -85,B 0,C 180,E1 27024.757,E2 27024.757} C_VEL
LIN {X 0,Y 556.25,Z 990.46,A -85,B 0,C 180,E1 27024.323,E2 27024.323} C_VEL
LIN {X 0,Y 555.942,Z 1006.691,A -85,B 0,C 180,E1 27023.699,E2 27023.699} C_VEL
LIN {X 0,Y 555.529,Z 1022.289,A -85,B 0,C 180,E1 27022.875,E2 27022.875} C_VEL
LIN {X 0,Y 555.085,Z 1036.242,A -85,B 0,C 180,E1 27021.93,E2 27021.93} C_VEL
LIN {X 0,Y 554.563,Z 1049.986,A -85,B 0,C 180,E1 27020.747,E2 27020.747} C_VEL
LIN {X 0,Y 554.099,Z 1061.507,A -85,B 0,C 180,E1 27019.499,E2 27019.499} C_VEL
LIN {X 0,Y 553.67,Z 1071.903,A -85,B 0,C 180,E1 27018.094,E2 27018.094} C_VEL
LIN {X 0,Y 553.334,Z 1080.556,A -85,B 0,C 180,E1 27016.587,E2 27016.587} C_VEL
LIN {X 0,Y 553.118,Z 1087.208,A -85,B 0,C 180,E1 27015.086,E2 27015.086} C_VEL
LIN {X 0,Y 552.973,Z 1091.978,A -85,B 0,C 180,E1 27013.593,E2 27013.593} C_VEL
LIN {X 0,Y 552.897,Z 1095.587,A -85,B 0,C 180,E1 27011.895,E2 27011.895} C_VEL
LIN {X 0,Y 552.901,Z 1097.168,A -85,B 0,C 180,E1 27010.311,E2 27010.311} C_VEL
LIN {X 0,Y 552.976,Z 1097.06,A -85,B 0,C 180,E1 27008.629,E2 27008.629} C_VEL
LIN {X 0,Y 553.108,Z 1095.285,A -85,B 0,C 180,E1 27007.059,E2 27007.059} C_VEL
LIN {X 0,Y 553.343,Z 1091.459,A -85,B 0,C 180,E1 27005.369,E2 27005.369} C_VEL
LIN {X 0,Y 553.653,Z 1086.167,A -85,B 0,C 180,E1 27003.829,E2 27003.829} C_VEL
LIN {X 0,Y 554.068,Z 1078.785,A -85,B 0,C 180,E1 27002.273,E2 27002.273} C_VEL
LIN {X 0,Y 554.546,Z 1070.556,A -85,B 0,C 180,E1 27000.928,E2 27000.928} C_VEL
LIN {X 0,Y 555.127,Z 1060.115,A -85,B 0,C 180,E1 26999.585,E2 26999.585} C_VEL
LIN {X 0,Y 555.711,Z 1048.596,A -85,B 0,C 180,E1 26998.4,E2 26998.4} C_VEL
LIN {X 0,Y 556.314,Z 1034.659,A -85,B 0,C 180,E1 26997.268,E2 26997.268} C_VEL
LIN {X 0,Y 556.761,Z 1020.931,A -85,B 0,C 180,E1 26996.394,E2 26996.394} C_VEL
LIN {X 0,Y 557.118,Z 1007.286,A -85,B 0,C 180,E1 26995.726,E2 26995.726} C_VEL
LIN {X 0,Y 557.368,Z 994.25,A -85,B 0,C 180,E1 26995.235,E2 26995.235} C_VEL
LIN {X 0,Y 557.506,Z 979.296,A -85,B 0,C 180,E1 26994.821,E2 26994.821} C_VEL
LIN {X 0,Y 557.905,Z 932.549,A -85,B 0,C 180,E1 26994.093,E2 26994.093} C_VEL
LIN {X 0,Y 559.773,Z 836.999,A -85,B 0,C 180,E1 26992.583,E2 26992.583} C_VEL
LIN {X 0,Y 560.814,Z 804.048,A -85,B 0,C 180,E1 26990.039,E2 26990.039} C_VEL
LIN {X 0,Y 561.671,Z 764.75,A -85,B 0,C 180,E1 26987.036,E2 26987.036} C_VEL
LIN {X 0,Y 562.523,Z 726.675,A -85,B 0,C 180,E1 26984.164,E2 26984.164} C_VEL
LIN {X 0,Y 563.086,Z 688.162,A -85,B 0,C 180,E1 26981.304,E2 26981.304} C_VEL
LIN {X 0,Y 563.379,Z 661.098,A -85,B 0,C 180,E1 26979.316,E2 26979.316} C_VEL
LIN {X 0,Y 558.377,Z 644.842,A -85,B 0,C 180,E1 26977.782,E2 26977.782} C_VEL
LIN {X 0,Y 553.47,Z 631.733,A -85,B 0,C 180,E1 26976.438,E2 26976.438} C_VEL
LIN {X 0,Y 553.501,Z 631.726,A -85,B 0,C 180,E1 26973.034,E2 26973.034} C_VEL
LIN {X 0,Y 553.511,Z 631.722,A -85,B 0,C 180,E1 26969.613,E2 26969.613} C_VEL
LIN {X 0,Y 553.488,Z 631.724,A -85,B 0,C 180,E1 26966.19,E2 26966.19} C_VEL
LIN {X 0,Y 553.472,Z 631.727,A -85,B 0,C 180,E1 26962.885,E2 26962.885} C_VEL
LIN {X 0,Y 553.488,Z 631.724,A -85,B 0,C 180,E1 26959.669,E2 26959.669} C_VEL
LIN {X 0,Y 553.495,Z 631.721,A -85,B 0,C 180,E1 26956.267,E2 26956.267} C_VEL
LIN {X 0,Y 553.491,Z 631.719,A -85,B 0,C 180,E1 26952.782,E2 26952.782} C_VEL
LIN {X 0,Y 553.481,Z 631.759,A -85,B 0,C 180,E1 26950.532,E2 26950.532} C_VEL
LIN {X 0,Y 561.503,Z 656.169,A -85,B 0,C 180,E1 26947.387,E2 26947.387} C_VEL
LIN {X 0,Y 568.2,Z 677.784,A -85,B 0,C 180,E1 26944.774,E2 26944.774} C_VEL
LIN {X 0,Y 568.334,Z 679.431,A -85,B 0,C 180,E1 26944.685,E2 26944.685} C_VEL
LIN {X 0,Y 576.402,Z 720.727,A -85,B 0,C 180,E1 26943.489,E2 26943.489} C_VEL
LIN {X 0,Y 570.518,Z 943.035,A -85,B 0,C 180,E1 26940.215,E2 26940.215} C_VEL
LIN {X 0,Y 569.383,Z 985.481,A -85,B 0,C 180,E1 26939.57,E2 26939.57} C_VEL
LIN {X 0,Y 568.302,Z 1007.606,A -85,B 0,C 180,E1 26939.061,E2 26939.061} C_VEL
LIN {X 0,Y 566.947,Z 1029.335,A -85,B 0,C 180,E1 26938.377,E2 26938.377} C_VEL
LIN {X 0,Y 565.356,Z 1051.376,A -85,B 0,C 180,E1 26937.489,E2 26937.489} C_VEL
LIN {X 0,Y 563.75,Z 1071.508,A -85,B 0,C 180,E1 26936.49,E2 26936.49} C_VEL
LIN {X 0,Y 561.974,Z 1091.659,A -85,B 0,C 180,E1 26935.277,E2 26935.277} C_VEL
LIN {X 0,Y 560.289,Z 1109.887,A -85,B 0,C 180,E1 26933.974,E2 26933.974} C_VEL
LIN {X 0,Y 558.599,Z 1127.932,A -85,B 0,C 180,E1 26932.466,E2 26932.466} C_VEL
LIN {X 0,Y 557.022,Z 1144.802,A -85,B 0,C 180,E1 26930.817,E2 26930.817} C_VEL
LIN {X 0,Y 555.608,Z 1160.453,A -85,B 0,C 180,E1 26929.008,E2 26929.008} C_VEL
LIN {X 0,Y 554.479,Z 1173.84,A -85,B 0,C 180,E1 26927.2,E2 26927.2} C_VEL
LIN {X 0,Y 553.571,Z 1186,A -85,B 0,C 180,E1 26925.289,E2 26925.289} C_VEL
LIN {X 0,Y 552.885,Z 1196.742,A -85,B 0,C 180,E1 26923.276,E2 26923.276} C_VEL
LIN {X 0,Y 552.408,Z 1206.053,A -85,B 0,C 180,E1 26921.166,E2 26921.166} C_VEL
LIN {X 0,Y 552.138,Z 1213.584,A -85,B 0,C 180,E1 26919.063,E2 26919.063} C_VEL
LIN {X 0,Y 551.999,Z 1219.434,A -85,B 0,C 180,E1 26916.945,E2 26916.945} C_VEL
LIN {X 0,Y 551.958,Z 1223.735,A -85,B 0,C 180,E1 26914.779,E2 26914.779} C_VEL
LIN {X 0,Y 551.964,Z 1226.411,A -85,B 0,C 180,E1 26912.698,E2 26912.698} C_VEL
LIN {X 0,Y 551.971,Z 1227.49,A -85,B 0,C 180,E1 26910.518,E2 26910.518} C_VEL
LIN {X 0,Y 551.977,Z 1226.943,A -85,B 0,C 180,E1 26908.234,E2 26908.234} C_VEL
LIN {X 0,Y 551.974,Z 1224.902,A -85,B 0,C 180,E1 26906.156,E2 26906.156} C_VEL
LIN {X 0,Y 551.99,Z 1221.059,A -85,B 0,C 180,E1 26903.968,E2 26903.968} C_VEL
LIN {X 0,Y 552.082,Z 1215.534,A -85,B 0,C 180,E1 26901.773,E2 26901.773} C_VEL
LIN {X 0,Y 552.262,Z 1208.888,A -85,B 0,C 180,E1 26899.779,E2 26899.779} C_VEL
LIN {X 0,Y 552.616,Z 1200.121,A -85,B 0,C 180,E1 26897.671,E2 26897.671} C_VEL
LIN {X 0,Y 553.159,Z 1189.99,A -85,B 0,C 180,E1 26895.661,E2 26895.661} C_VEL
LIN {X 0,Y 553.91,Z 1178.452,A -85,B 0,C 180,E1 26893.751,E2 26893.751} C_VEL
LIN {X 0,Y 554.897,Z 1164.818,A -85,B 0,C 180,E1 26891.835,E2 26891.835} C_VEL
LIN {X 0,Y 556.109,Z 1149.718,A -85,B 0,C 180,E1 26890.023,E2 26890.023} C_VEL
LIN {X 0,Y 557.461,Z 1133.636,A -85,B 0,C 180,E1 26888.37,E2 26888.37} C_VEL
LIN {X 0,Y 558.978,Z 1115.988,A -85,B 0,C 180,E1 26886.824,E2 26886.824} C_VEL
LIN {X 0,Y 560.626,Z 1096.77,A -85,B 0,C 180,E1 26885.388,E2 26885.388} C_VEL
LIN {X 0,Y 562.267,Z 1077.091,A -85,B 0,C 180,E1 26884.138,E2 26884.138} C_VEL
LIN {X 0,Y 563.965,Z 1055.734,A -85,B 0,C 180,E1 26883.006,E2 26883.006} C_VEL
LIN {X 0,Y 565.56,Z 1033.776,A -85,B 0,C 180,E1 26882.061,E2 26882.061} C_VEL
LIN {X 0,Y 567.025,Z 1011.163,A -85,B 0,C 180,E1 26881.286,E2 26881.286} C_VEL
LIN {X 0,Y 568.374,Z 987.492,A -85,B 0,C 180,E1 26880.673,E2 26880.673} C_VEL
LIN {X 0,Y 569.39,Z 961.996,A -85,B 0,C 180,E1 26880.208,E2 26880.208} C_VEL
LIN {X 0,Y 572.537,Z 867.698,A -85,B 0,C 180,E1 26878.664,E2 26878.664} C_VEL
LIN {X 0,Y 577.095,Z 773.581,A -85,B 0,C 180,E1 26876.972,E2 26876.972} C_VEL
LIN {X 0,Y 580.239,Z 719.713,A -85,B 0,C 180,E1 26875.928,E2 26875.928} C_VEL
LIN {X 0,Y 577.16,Z 695.178,A -85,B 0,C 180,E1 26874.955,E2 26874.955} C_VEL
LIN {X 0,Y 575.09,Z 683.21,A -85,B 0,C 180,E1 26874.363,E2 26874.363} C_VEL
LIN {X 0,Y 570.368,Z 672.874,A -85,B 0,C 180,E1 26873.452,E2 26873.452} C_VEL
LIN {X 0,Y 566.9,Z 665.99,A -85,B 0,C 180,E1 26872.701,E2 26872.701} C_VEL
LIN {X 0,Y 564.212,Z 657.478,A -85,B 0,C 180,E1 26871.013,E2 26871.013} C_VEL
LIN {X 0,Y 561.866,Z 651.164,A -85,B 0,C 180,E1 26869.456,E2 26869.456} C_VEL
LIN {X 0,Y 560.471,Z 647.638,A -85,B 0,C 180,E1 26868.376,E2 26868.376} C_VEL
LIN {X 0,Y 559.19,Z 644.424,A -85,B 0,C 180,E1 26867.151,E2 26867.151} C_VEL
LIN {X 0,Y 557.834,Z 640.852,A -85,B 0,C 180,E1 26865.07,E2 26865.07} C_VEL
LIN {X 0,Y 557.122,Z 639.997,A -85,B 0,C 180,E1 26863.074,E2 26863.074} C_VEL
LIN {X 0,Y 557.742,Z 640.818,A -85,B 0,C 180,E1 26861.145,E2 26861.145} C_VEL
LIN {X 0,Y 559.126,Z 644.403,A -85,B 0,C 180,E1 26858.929,E2 26858.929} C_VEL
LIN {X 0,Y 559.752,Z 646.023,A -85,B 0,C 180,E1 26858.353,E2 26858.353} C_VEL
LIN {X 0,Y 563.977,Z 651.23,A -85,B 0,C 180,E1 26857.327,E2 26857.327} C_VEL
LIN {X 0,Y 567.751,Z 656.24,A -85,B 0,C 180,E1 26856.533,E2 26856.533} C_VEL
LIN {X 0,Y 573.068,Z 663.812,A -85,B 0,C 180,E1 26855.532,E2 26855.532} C_VEL
LIN {X 0,Y 579.801,Z 675.216,A -85,B 0,C 180,E1 26854.391,E2 26854.391} C_VEL
LIN {X 0,Y 582.107,Z 680.076,A -85,B 0,C 180,E1 26854.015,E2 26854.015} C_VEL
LIN {X 0,Y 576.306,Z 770.852,A -85,B 0,C 180,E1 26852.274,E2 26852.274} C_VEL
LIN {X 0,Y 572.16,Z 859.749,A -85,B 0,C 180,E1 26850.698,E2 26850.698} C_VEL
LIN {X 0,Y 569.427,Z 939.289,A -85,B 0,C 180,E1 26849.365,E2 26849.365} C_VEL
LIN {X 0,Y 568.422,Z 962.398,A -85,B 0,C 180,E1 26848.788,E2 26848.788} C_VEL
LIN {X 0,Y 567.151,Z 984.226,A -85,B 0,C 180,E1 26848.052,E2 26848.052} C_VEL
LIN {X 0,Y 565.685,Z 1005.706,A -85,B 0,C 180,E1 26847.133,E2 26847.133} C_VEL
LIN {X 0,Y 564.043,Z 1026.861,A -85,B 0,C 180,E1 26846.02,E2 26846.02} C_VEL
LIN {X 0,Y 562.41,Z 1046.018,A -85,B 0,C 180,E1 26844.81,E2 26844.81} C_VEL
LIN {X 0,Y 560.674,Z 1065.035,A -85,B 0,C 180,E1 26843.38,E2 26843.38} C_VEL
LIN {X 0,Y 558.978,Z 1082.515,A -85,B 0,C 180,E1 26841.815,E2 26841.815} C_VEL
LIN {X 0,Y 557.506,Z 1097.457,A -85,B 0,C 180,E1 26840.254,E2 26840.254} C_VEL
LIN {X 0,Y 556.179,Z 1111.498,A -85,B 0,C 180,E1 26838.557,E2 26838.557} C_VEL
LIN {X 0,Y 554.938,Z 1124.845,A -85,B 0,C 180,E1 26836.65,E2 26836.65} C_VEL
LIN {X 0,Y 553.964,Z 1136.099,A -85,B 0,C 180,E1 26834.746,E2 26834.746} C_VEL
LIN {X 0,Y 553.226,Z 1146.104,A -85,B 0,C 180,E1 26832.74,E2 26832.74} C_VEL
LIN {X 0,Y 552.674,Z 1154.703,A -85,B 0,C 180,E1 26830.636,E2 26830.636} C_VEL
LIN {X 0,Y 552.322,Z 1161.485,A -85,B 0,C 180,E1 26828.539,E2 26828.539} C_VEL
LIN {X 0,Y 552.121,Z 1166.934,A -85,B 0,C 180,E1 26826.345,E2 26826.345} C_VEL
LIN {X 0,Y 552.024,Z 1170.533,A -85,B 0,C 180,E1 26824.261,E2 26824.261} C_VEL
LIN {X 0,Y 551.981,Z 1172.74,A -85,B 0,C 180,E1 26822.078,E2 26822.078} C_VEL
LIN {X 0,Y 551.982,Z 1173.467,A -85,B 0,C 180,E1 26819.898,E2 26819.898} C_VEL
LIN {X 0,Y 551.976,Z 1172.528,A -85,B 0,C 180,E1 26817.718,E2 26817.718} C_VEL
LIN {X 0,Y 552.021,Z 1169.926,A -85,B 0,C 180,E1 26815.431,E2 26815.431} C_VEL
LIN {X 0,Y 552.122,Z 1165.863,A -85,B 0,C 180,E1 26813.242,E2 26813.242} C_VEL
LIN {X 0,Y 552.32,Z 1160.01,A -85,B 0,C 180,E1 26811.046,E2 26811.046} C_VEL
LIN {X 0,Y 552.704,Z 1152.386,A -85,B 0,C 180,E1 26808.841,E2 26808.841} C_VEL
LIN {X 0,Y 553.288,Z 1143.338,A -85,B 0,C 180,E1 26806.734,E2 26806.734} C_VEL
LIN {X 0,Y 554.079,Z 1132.858,A -85,B 0,C 180,E1 26804.727,E2 26804.727} C_VEL
LIN {X 0,Y 555.08,Z 1121.01,A -85,B 0,C 180,E1 26802.82,E2 26802.82} C_VEL
LIN {X 0,Y 556.314,Z 1107.652,A -85,B 0,C 180,E1 26800.982,E2 26800.982} C_VEL
LIN {X 0,Y 557.783,Z 1092.584,A -85,B 0,C 180,E1 26799.213,E2 26799.213} C_VEL
LIN {X 0,Y 559.327,Z 1076.615,A -85,B 0,C 180,E1 26797.621,E2 26797.621} C_VEL
LIN {X 0,Y 561.045,Z 1058.839,A -85,B 0,C 180,E1 26796.103,E2 26796.103} C_VEL
LIN {X 0,Y 562.771,Z 1040.441,A -85,B 0,C 180,E1 26794.763,E2 26794.763} C_VEL
LIN {X 0,Y 564.453,Z 1020.82,A -85,B 0,C 180,E1 26793.564,E2 26793.564} C_VEL
LIN {X 0,Y 566.023,Z 1000.739,A -85,B 0,C 180,E1 26792.548,E2 26792.548} C_VEL
LIN {X 0,Y 567.513,Z 979.158,A -85,B 0,C 180,E1 26791.658,E2 26791.658} C_VEL
LIN {X 0,Y 568.74,Z 957.381,A -85,B 0,C 180,E1 26790.95,E2 26790.95} C_VEL
LIN {X 0,Y 569.727,Z 934.9,A -85,B 0,C 180,E1 26790.422,E2 26790.422} C_VEL
LIN {X 0,Y 570.688,Z 899.021,A -85,B 0,C 180,E1 26789.864,E2 26789.864} C_VEL
LIN {X 0,Y 576.367,Z 684.308,A -85,B 0,C 180,E1 26786.715,E2 26786.715} C_VEL
LIN {X 0,Y 576.451,Z 675.327,A -85,B 0,C 180,E1 26786.569,E2 26786.569} C_VEL
LIN {X 0,Y 564.056,Z 651.315,A -85,B 0,C 180,E1 26785.384,E2 26785.384} C_VEL
LIN {X 0,Y 554.718,Z 635.091,A -85,B 0,C 180,E1 26784.474,E2 26784.474} C_VEL
LIN {X 0,Y 553.476,Z 631.727,A -85,B 0,C 180,E1 26784.305,E2 26784.305} C_VEL
LIN {X 0,Y 553.505,Z 631.724,A -85,B 0,C 180,E1 26781.053,E2 26781.053} C_VEL
LIN {X 0,Y 553.497,Z 631.721,A -85,B 0,C 180,E1 26777.635,E2 26777.635} C_VEL
LIN {X 0,Y 553.492,Z 631.72,A -85,B 0,C 180,E1 26774.33,E2 26774.33} C_VEL
LIN {X 0,Y 553.433,Z 631.729,A -85,B 0,C 180,E1 26771.119,E2 26771.119} C_VEL
LIN {X 0,Y 553.472,Z 631.726,A -85,B 0,C 180,E1 26769.881,E2 26769.881} C_VEL
LIN {X 0,Y 552.419,Z 631.863,A -85,B 0,C 180,E1 26769.084,E2 26769.084} C_VEL
LIN {X 0,Y 546.05,Z 632.659,A -85,B 0,C 180,E1 26766.845,E2 26766.845} C_VEL
LIN {X 0,Y 545.556,Z 632.713,A -85,B 0,C 180,E1 26766.262,E2 26766.262} C_VEL
LIN {X 0,Y 545.543,Z 632.714,A -85,B 0,C 180,E1 26762.925,E2 26762.925} C_VEL
LIN {X 0,Y 545.559,Z 632.708,A -85,B 0,C 180,E1 26759.482,E2 26759.482} C_VEL
LIN {X 0,Y 545.53,Z 632.709,A -85,B 0,C 180,E1 26756.215,E2 26756.215} C_VEL
LIN {X 0,Y 545.493,Z 632.714,A -85,B 0,C 180,E1 26752.789,E2 26752.789} C_VEL
LIN {X 0,Y 545.548,Z 632.711,A -85,B 0,C 180,E1 26749.487,E2 26749.487} C_VEL
LIN {X 0,Y 545.548,Z 632.713,A -85,B 0,C 180,E1 26746.177,E2 26746.177} C_VEL
LIN {X 0,Y 545.549,Z 632.703,A -85,B 0,C 180,E1 26742.814,E2 26742.814} C_VEL
LIN {X 0,Y 545.548,Z 632.706,A -85,B 0,C 180,E1 26739.496,E2 26739.496} C_VEL
LIN {X 0,Y 545.506,Z 632.716,A -85,B 0,C 180,E1 26736.21,E2 26736.21} C_VEL
LIN {X 0,Y 545.529,Z 632.705,A -85,B 0,C 180,E1 26732.943,E2 26732.943} C_VEL
LIN {X 0,Y 545.529,Z 632.715,A -85,B 0,C 180,E1 26729.686,E2 26729.686} C_VEL
LIN {X 0,Y 545.539,Z 632.701,A -85,B 0,C 180,E1 26726.323,E2 26726.323} C_VEL
LIN {X 0,Y 545.559,Z 632.707,A -85,B 0,C 180,E1 26722.948,E2 26722.948} C_VEL
LIN {X 0,Y 545.515,Z 632.701,A -85,B 0,C 180,E1 26719.547,E2 26719.547} C_VEL
LIN {X 0,Y 545.514,Z 632.716,A -85,B 0,C 180,E1 26716.217,E2 26716.217} C_VEL
LIN {X 0,Y 545.536,Z 632.714,A -85,B 0,C 180,E1 26712.949,E2 26712.949} C_VEL
LIN {X 0,Y 545.532,Z 632.711,A -85,B 0,C 180,E1 26709.622,E2 26709.622} C_VEL
LIN {X 0,Y 545.564,Z 632.705,A -85,B 0,C 180,E1 26706.223,E2 26706.223} C_VEL
LIN {X 0,Y 545.53,Z 632.712,A -85,B 0,C 180,E1 26702.848,E2 26702.848} C_VEL
LIN {X 0,Y 545.509,Z 632.717,A -85,B 0,C 180,E1 26699.477,E2 26699.477} C_VEL
LIN {X 0,Y 545.548,Z 632.715,A -85,B 0,C 180,E1 26696.142,E2 26696.142} C_VEL
LIN {X 0,Y 545.535,Z 632.715,A -85,B 0,C 180,E1 26692.785,E2 26692.785} C_VEL
LIN {X 0,Y 545.549,Z 632.711,A -85,B 0,C 180,E1 26689.412,E2 26689.412} C_VEL
LIN {X 0,Y 545.548,Z 632.711,A -85,B 0,C 180,E1 26686.074,E2 26686.074} C_VEL
LIN {X 0,Y 545.585,Z 632.953,A -85,B 0,C 180,E1 26683.24,E2 26683.24} C_VEL
LIN {X 0,Y 553.124,Z 659.768,A -85,B 0,C 180,E1 26680.694,E2 26680.694} C_VEL
LIN {X 0,Y 554.285,Z 664.904,A -85,B 0,C 180,E1 26680.222,E2 26680.222} C_VEL
LIN {X 0,Y 553.173,Z 708.869,A -85,B 0,C 180,E1 26676.745,E2 26676.745} C_VEL
LIN {X 0,Y 552.091,Z 750.193,A -85,B 0,C 180,E1 26673.466,E2 26673.466} C_VEL
LIN {X 0,Y 550.953,Z 790.912,A -85,B 0,C 180,E1 26670.251,E2 26670.251} C_VEL
LIN {X 0,Y 549.986,Z 831.6,A -85,B 0,C 180,E1 26667.068,E2 26667.068} C_VEL
LIN {X 0,Y 550.225,Z 839.944,A -85,B 0,C 180,E1 26666.932,E2 26666.932} C_VEL
LIN {X 0,Y 548.585,Z 974.823,A -85,B 0,C 180,E1 26664.915,E2 26664.915} C_VEL
LIN {X 0,Y 548.418,Z 991.234,A -85,B 0,C 180,E1 26664.477,E2 26664.477} C_VEL
LIN {X 0,Y 548.102,Z 1007.316,A -85,B 0,C 180,E1 26663.851,E2 26663.851} C_VEL
LIN {X 0,Y 547.697,Z 1022.206,A -85,B 0,C 180,E1 26663.063,E2 26663.063} C_VEL
LIN {X 0,Y 547.24,Z 1036.352,A -85,B 0,C 180,E1 26662.107,E2 26662.107} C_VEL
LIN {X 0,Y 546.708,Z 1049.838,A -85,B 0,C 180,E1 26660.947,E2 26660.947} C_VEL
LIN {X 0,Y 546.268,Z 1060.729,A -85,B 0,C 180,E1 26659.79,E2 26659.79} C_VEL
LIN {X 0,Y 545.81,Z 1071.223,A -85,B 0,C 180,E1 26658.395,E2 26658.395} C_VEL
LIN {X 0,Y 545.465,Z 1079.929,A -85,B 0,C 180,E1 26656.943,E2 26656.943} C_VEL
LIN {X 0,Y 545.193,Z 1087.356,A -85,B 0,C 180,E1 26655.311,E2 26655.311} C_VEL
LIN {X 0,Y 545.047,Z 1092.447,A -85,B 0,C 180,E1 26653.795,E2 26653.795} C_VEL
LIN {X 0,Y 544.95,Z 1096.404,A -85,B 0,C 180,E1 26651.964,E2 26651.964} C_VEL
LIN {X 0,Y 544.957,Z 1098.102,A -85,B 0,C 180,E1 26650.356,E2 26650.356} C_VEL
LIN {X 0,Y 545.04,Z 1098.044,A -85,B 0,C 180,E1 26648.596,E2 26648.596} C_VEL
LIN {X 0,Y 545.191,Z 1096.199,A -85,B 0,C 180,E1 26646.95,E2 26646.95} C_VEL
LIN {X 0,Y 545.448,Z 1092.407,A -85,B 0,C 180,E1 26645.257,E2 26645.257} C_VEL
LIN {X 0,Y 545.791,Z 1087.014,A -85,B 0,C 180,E1 26643.674,E2 26643.674} C_VEL
LIN {X 0,Y 546.265,Z 1079.345,A -85,B 0,C 180,E1 26642.046,E2 26642.046} C_VEL
LIN {X 0,Y 546.804,Z 1070.554,A -85,B 0,C 180,E1 26640.626,E2 26640.626} C_VEL
LIN {X 0,Y 547.439,Z 1059.883,A -85,B 0,C 180,E1 26639.265,E2 26639.265} C_VEL
LIN {X 0,Y 548.064,Z 1047.959,A -85,B 0,C 180,E1 26638.064,E2 26638.064} C_VEL
LIN {X 0,Y 548.645,Z 1035.056,A -85,B 0,C 180,E1 26637.02,E2 26637.02} C_VEL
LIN {X 0,Y 549.119,Z 1021.09,A -85,B 0,C 180,E1 26636.135,E2 26636.135} C_VEL
LIN {X 0,Y 549.472,Z 1008.451,A -85,B 0,C 180,E1 26635.51,E2 26635.51} C_VEL
LIN {X 0,Y 549.743,Z 995.345,A -85,B 0,C 180,E1 26635.006,E2 26635.006} C_VEL
LIN {X 0,Y 549.899,Z 980.513,A -85,B 0,C 180,E1 26634.585,E2 26634.585} C_VEL
LIN {X 0,Y 550.229,Z 940.159,A -85,B 0,C 180,E1 26633.936,E2 26633.936} C_VEL
LIN {X 0,Y 552.307,Z 838.315,A -85,B 0,C 180,E1 26632.299,E2 26632.299} C_VEL
LIN {X 0,Y 553.273,Z 811.448,A -85,B 0,C 180,E1 26630.217,E2 26630.217} C_VEL
LIN {X 0,Y 554.321,Z 769.383,A -85,B 0,C 180,E1 26626.967,E2 26626.967} C_VEL
LIN {X 0,Y 555.311,Z 728.262,A -85,B 0,C 180,E1 26623.846,E2 26623.846} C_VEL
LIN {X 0,Y 556.121,Z 682.314,A -85,B 0,C 180,E1 26620.407,E2 26620.407} C_VEL
LIN {X 0,Y 556.479,Z 664.644,A -85,B 0,C 180,E1 26619.116,E2 26619.116} C_VEL
LIN {X 0,Y 551.615,Z 648.646,A -85,B 0,C 180,E1 26617.58,E2 26617.58} C_VEL
LIN {X 0,Y 546.396,Z 635.458,A -85,B 0,C 180,E1 26616.198,E2 26616.198} C_VEL
LIN {X 0,Y 545.555,Z 632.721,A -85,B 0,C 180,E1 26615.908,E2 26615.908} C_VEL
LIN {X 0,Y 545.541,Z 632.716,A -85,B 0,C 180,E1 26612.608,E2 26612.608} C_VEL
LIN {X 0,Y 545.565,Z 632.711,A -85,B 0,C 180,E1 26609,E2 26609} C_VEL
LIN {X 0,Y 545.565,Z 632.711,A -85,B 0,C 180,E1 26605.504,E2 26605.504} C_VEL
LIN {X 0,Y 545.544,Z 632.713,A -85,B 0,C 180,E1 26602.119,E2 26602.119} C_VEL
LIN {X 0,Y 545.537,Z 632.713,A -85,B 0,C 180,E1 26598.851,E2 26598.851} C_VEL
LIN {X 0,Y 545.55,Z 632.714,A -85,B 0,C 180,E1 26595.56,E2 26595.56} C_VEL
LIN {X 0,Y 545.559,Z 632.708,A -85,B 0,C 180,E1 26592.126,E2 26592.126} C_VEL
LIN {X 0,Y 545.599,Z 632.89,A -85,B 0,C 180,E1 26590.999,E2 26590.999} C_VEL
LIN {X 0,Y 554.146,Z 658.805,A -85,B 0,C 180,E1 26587.614,E2 26587.614} C_VEL
LIN {X 0,Y 560.267,Z 678.488,A -85,B 0,C 180,E1 26585.219,E2 26585.219} C_VEL
LIN {X 0,Y 561.829,Z 682.512,A -85,B 0,C 180,E1 26585.047,E2 26585.047} C_VEL
LIN {X 0,Y 569.482,Z 722.13,A -85,B 0,C 180,E1 26583.878,E2 26583.878} C_VEL
LIN {X 0,Y 563.219,Z 947.139,A -85,B 0,C 180,E1 26580.509,E2 26580.509} C_VEL
LIN {X 0,Y 562.081,Z 985.979,A -85,B 0,C 180,E1 26579.897,E2 26579.897} C_VEL
LIN {X 0,Y 560.924,Z 1008.641,A -85,B 0,C 180,E1 26579.363,E2 26579.363} C_VEL
LIN {X 0,Y 559.488,Z 1030.417,A -85,B 0,C 180,E1 26578.657,E2 26578.657} C_VEL
LIN {X 0,Y 557.868,Z 1051.812,A -85,B 0,C 180,E1 26577.773,E2 26577.773} C_VEL
LIN {X 0,Y 556.204,Z 1071.813,A -85,B 0,C 180,E1 26576.762,E2 26576.762} C_VEL
LIN {X 0,Y 554.362,Z 1091.932,A -85,B 0,C 180,E1 26575.534,E2 26575.534} C_VEL
LIN {X 0,Y 552.594,Z 1110.278,A -85,B 0,C 180,E1 26574.198,E2 26574.198} C_VEL
LIN {X 0,Y 550.739,Z 1129.184,A -85,B 0,C 180,E1 26572.579,E2 26572.579} C_VEL
LIN {X 0,Y 549.213,Z 1144.844,A -85,B 0,C 180,E1 26571.016,E2 26571.016} C_VEL
LIN {X 0,Y 547.823,Z 1159.62,A -85,B 0,C 180,E1 26569.289,E2 26569.289} C_VEL
LIN {X 0,Y 546.629,Z 1173.126,A -85,B 0,C 180,E1 26567.455,E2 26567.455} C_VEL
LIN {X 0,Y 545.669,Z 1185.373,A -85,B 0,C 180,E1 26565.516,E2 26565.516} C_VEL
LIN {X 0,Y 544.939,Z 1196.179,A -85,B 0,C 180,E1 26563.469,E2 26563.469} C_VEL
LIN {X 0,Y 544.432,Z 1205.525,A -85,B 0,C 180,E1 26561.331,E2 26561.331} C_VEL
LIN {X 0,Y 544.149,Z 1213.115,A -85,B 0,C 180,E1 26559.197,E2 26559.197} C_VEL
LIN {X 0,Y 544.01,Z 1218.929,A -85,B 0,C 180,E1 26557.072,E2 26557.072} C_VEL
LIN {X 0,Y 543.962,Z 1223.323,A -85,B 0,C 180,E1 26554.849,E2 26554.849} C_VEL
LIN {X 0,Y 543.97,Z 1226.01,A -85,B 0,C 180,E1 26552.738,E2 26552.738} C_VEL
LIN {X 0,Y 543.981,Z 1227.096,A -85,B 0,C 180,E1 26550.525,E2 26550.525} C_VEL
LIN {X 0,Y 543.987,Z 1226.543,A -85,B 0,C 180,E1 26548.208,E2 26548.208} C_VEL
LIN {X 0,Y 543.981,Z 1224.486,A -85,B 0,C 180,E1 26546.099,E2 26546.099} C_VEL
LIN {X 0,Y 543.998,Z 1220.613,A -85,B 0,C 180,E1 26543.879,E2 26543.879} C_VEL
LIN {X 0,Y 544.096,Z 1215.056,A -85,B 0,C 180,E1 26541.651,E2 26541.651} C_VEL
LIN {X 0,Y 544.295,Z 1207.999,A -85,B 0,C 180,E1 26539.52,E2 26539.52} C_VEL
LIN {X 0,Y 544.681,Z 1199.068,A -85,B 0,C 180,E1 26537.381,E2 26537.381} C_VEL
LIN {X 0,Y 545.272,Z 1188.772,A -85,B 0,C 180,E1 26535.34,E2 26535.34} C_VEL
LIN {X 0,Y 546.076,Z 1177.113,A -85,B 0,C 180,E1 26533.402,E2 26533.402} C_VEL
LIN {X 0,Y 547.09,Z 1163.931,A -85,B 0,C 180,E1 26531.544,E2 26531.544} C_VEL
LIN {X 0,Y 548.4,Z 1148.509,A -85,B 0,C 180,E1 26529.682,E2 26529.682} C_VEL
LIN {X 0,Y 549.859,Z 1132.264,A -85,B 0,C 180,E1 26527.999,E2 26527.999} C_VEL
LIN {X 0,Y 551.518,Z 1113.801,A -85,B 0,C 180,E1 26526.379,E2 26526.379} C_VEL
LIN {X 0,Y 553.228,Z 1095.055,A -85,B 0,C 180,E1 26524.979,E2 26524.979} C_VEL
LIN {X 0,Y 554.997,Z 1074.737,A -85,B 0,C 180,E1 26523.691,E2 26523.691} C_VEL
LIN {X 0,Y 556.693,Z 1054.755,A -85,B 0,C 180,E1 26522.624,E2 26522.624} C_VEL
LIN {X 0,Y 558.378,Z 1032.822,A -85,B 0,C 180,E1 26521.67,E2 26521.67} C_VEL
LIN {X 0,Y 559.959,Z 1010.101,A -85,B 0,C 180,E1 26520.882,E2 26520.882} C_VEL
LIN {X 0,Y 561.401,Z 986.158,A -85,B 0,C 180,E1 26520.255,E2 26520.255} C_VEL
LIN {X 0,Y 562.55,Z 958.974,A -85,B 0,C 180,E1 26519.754,E2 26519.754} C_VEL
LIN {X 0,Y 565.948,Z 867.812,A -85,B 0,C 180,E1 26518.206,E2 26518.206} C_VEL
LIN {X 0,Y 570.991,Z 773.809,A -85,B 0,C 180,E1 26516.455,E2 26516.455} C_VEL
LIN {X 0,Y 574.386,Z 721.281,A -85,B 0,C 180,E1 26515.401,E2 26515.401} C_VEL
LIN {X 0,Y 571.789,Z 698.142,A -85,B 0,C 180,E1 26514.442,E2 26514.442} C_VEL
LIN {X 0,Y 570.043,Z 687.561,A -85,B 0,C 180,E1 26513.908,E2 26513.908} C_VEL
LIN {X 0,Y 565.446,Z 677.303,A -85,B 0,C 180,E1 26512.937,E2 26512.937} C_VEL
LIN {X 0,Y 561.998,Z 670.623,A -85,B 0,C 180,E1 26512.161,E2 26512.161} C_VEL
LIN {X 0,Y 558.608,Z 664.237,A -85,B 0,C 180,E1 26511.301,E2 26511.301} C_VEL
LIN {X 0,Y 556.329,Z 657.313,A -85,B 0,C 180,E1 26509.648,E2 26509.648} C_VEL
LIN {X 0,Y 554.358,Z 652.54,A -85,B 0,C 180,E1 26508.135,E2 26508.135} C_VEL
LIN {X 0,Y 553.328,Z 649.815,A -85,B 0,C 180,E1 26507.044,E2 26507.044} C_VEL
LIN {X 0,Y 552.061,Z 646.376,A -85,B 0,C 180,E1 26504.942,E2 26504.942} C_VEL
LIN {X 0,Y 551.451,Z 645.631,A -85,B 0,C 180,E1 26502.9,E2 26502.9} C_VEL
LIN {X 0,Y 552.04,Z 646.677,A -85,B 0,C 180,E1 26500.948,E2 26500.948} C_VEL
LIN {X 0,Y 552.52,Z 648.352,A -85,B 0,C 180,E1 26499.943,E2 26499.943} C_VEL
LIN {X 0,Y 556.834,Z 653.122,A -85,B 0,C 180,E1 26498.591,E2 26498.591} C_VEL
LIN {X 0,Y 560.899,Z 658.361,A -85,B 0,C 180,E1 26497.548,E2 26497.548} C_VEL
LIN {X 0,Y 564.444,Z 663.265,A -85,B 0,C 180,E1 26496.76,E2 26496.76} C_VEL
LIN {X 0,Y 569.235,Z 670.329,A -85,B 0,C 180,E1 26495.81,E2 26495.81} C_VEL
LIN {X 0,Y 575.265,Z 680.853,A -85,B 0,C 180,E1 26494.73,E2 26494.73} C_VEL
LIN {X 0,Y 576.36,Z 683.563,A -85,B 0,C 180,E1 26494.526,E2 26494.526} C_VEL
LIN {X 0,Y 569.958,Z 774.729,A -85,B 0,C 180,E1 26492.719,E2 26492.719} C_VEL
LIN {X 0,Y 565.447,Z 862.607,A -85,B 0,C 180,E1 26491.108,E2 26491.108} C_VEL
LIN {X 0,Y 562.509,Z 939.969,A -85,B 0,C 180,E1 26489.766,E2 26489.766} C_VEL
LIN {X 0,Y 561.43,Z 963.036,A -85,B 0,C 180,E1 26489.177,E2 26489.177} C_VEL
LIN {X 0,Y 560.025,Z 985.64,A -85,B 0,C 180,E1 26488.397,E2 26488.397} C_VEL
LIN {X 0,Y 558.491,Z 1006.687,A -85,B 0,C 180,E1 26487.476,E2 26487.476} C_VEL
LIN {X 0,Y 556.812,Z 1027.125,A -85,B 0,C 180,E1 26486.384,E2 26486.384} C_VEL
LIN {X 0,Y 555.089,Z 1046.284,A -85,B 0,C 180,E1 26485.16,E2 26485.16} C_VEL
LIN {X 0,Y 553.281,Z 1065.013,A -85,B 0,C 180,E1 26483.735,E2 26483.735} C_VEL
LIN {X 0,Y 551.54,Z 1081.928,A -85,B 0,C 180,E1 26482.211,E2 26482.211} C_VEL
LIN {X 0,Y 549.901,Z 1097.828,A -85,B 0,C 180,E1 26480.538,E2 26480.538} C_VEL
LIN {X 0,Y 548.496,Z 1111.828,A -85,B 0,C 180,E1 26478.826,E2 26478.826} C_VEL
LIN {X 0,Y 547.175,Z 1125.189,A -85,B 0,C 180,E1 26476.893,E2 26476.893} C_VEL
LIN {X 0,Y 546.138,Z 1136.463,A -85,B 0,C 180,E1 26474.962,E2 26474.962} C_VEL
LIN {X 0,Y 545.345,Z 1146.491,A -85,B 0,C 180,E1 26472.928,E2 26472.928} C_VEL
LIN {X 0,Y 544.747,Z 1155.093,A -85,B 0,C 180,E1 26470.793,E2 26470.793} C_VEL
LIN {X 0,Y 544.366,Z 1161.893,A -85,B 0,C 180,E1 26468.665,E2 26468.665} C_VEL
LIN {X 0,Y 544.148,Z 1167.348,A -85,B 0,C 180,E1 26466.438,E2 26466.438} C_VEL
LIN {X 0,Y 544.042,Z 1170.944,A -85,B 0,C 180,E1 26464.324,E2 26464.324} C_VEL
LIN {X 0,Y 543.993,Z 1173.149,A -85,B 0,C 180,E1 26462.109,E2 26462.109} C_VEL
LIN {X 0,Y 543.993,Z 1173.861,A -85,B 0,C 180,E1 26459.897,E2 26459.897} C_VEL
LIN {X 0,Y 543.987,Z 1172.905,A -85,B 0,C 180,E1 26457.685,E2 26457.685} C_VEL
LIN {X 0,Y 544.035,Z 1170.269,A -85,B 0,C 180,E1 26455.364,E2 26455.364} C_VEL
LIN {X 0,Y 544.145,Z 1166.161,A -85,B 0,C 180,E1 26453.143,E2 26453.143} C_VEL
LIN {X 0,Y 544.358,Z 1160.27,A -85,B 0,C 180,E1 26450.914,E2 26450.914} C_VEL
LIN {X 0,Y 544.772,Z 1152.583,A -85,B 0,C 180,E1 26448.677,E2 26448.677} C_VEL
LIN {X 0,Y 545.39,Z 1143.465,A -85,B 0,C 180,E1 26446.539,E2 26446.539} C_VEL
LIN {X 0,Y 546.232,Z 1132.928,A -85,B 0,C 180,E1 26444.502,E2 26444.502} C_VEL
LIN {X 0,Y 547.291,Z 1120.978,A -85,B 0,C 180,E1 26442.568,E2 26442.568} C_VEL
LIN {X 0,Y 548.643,Z 1106.922,A -85,B 0,C 180,E1 26440.631,E2 26440.631} C_VEL
LIN {X 0,Y 550.181,Z 1091.827,A -85,B 0,C 180,E1 26438.857,E2 26438.857} C_VEL
LIN {X 0,Y 551.887,Z 1075.102,A -85,B 0,C 180,E1 26437.19,E2 26437.19} C_VEL
LIN {X 0,Y 553.644,Z 1057.393,A -85,B 0,C 180,E1 26435.687,E2 26435.687} C_VEL
LIN {X 0,Y 555.51,Z 1038.044,A -85,B 0,C 180,E1 26434.295,E2 26434.295} C_VEL
LIN {X 0,Y 557.226,Z 1018.674,A -85,B 0,C 180,E1 26433.119,E2 26433.119} C_VEL
LIN {X 0,Y 558.893,Z 997.884,A -85,B 0,C 180,E1 26432.084,E2 26432.084} C_VEL
LIN {X 0,Y 560.353,Z 976.655,A -85,B 0,C 180,E1 26431.23,E2 26431.23} C_VEL
LIN {X 0,Y 561.616,Z 954.255,A -85,B 0,C 180,E1 26430.526,E2 26430.526} C_VEL
LIN {X 0,Y 562.626,Z 931.988,A -85,B 0,C 180,E1 26430.014,E2 26430.014} C_VEL
LIN {X 0,Y 569.694,Z 678.279,A -85,B 0,C 180,E1 26426.208,E2 26426.208} C_VEL
LIN {X 0,Y 558.11,Z 655.77,A -85,B 0,C 180,E1 26425.072,E2 26425.072} C_VEL
LIN {X 0,Y 546.834,Z 636.221,A -85,B 0,C 180,E1 26423.966,E2 26423.966} C_VEL
LIN {X 0,Y 545.51,Z 632.715,A -85,B 0,C 180,E1 26423.807,E2 26423.807} C_VEL
LIN {X 0,Y 545.569,Z 632.706,A -85,B 0,C 180,E1 26420.498,E2 26420.498} C_VEL
LIN {X 0,Y 545.554,Z 632.713,A -85,B 0,C 180,E1 26417.15,E2 26417.15} C_VEL
LIN {X 0,Y 545.561,Z 632.712,A -85,B 0,C 180,E1 26413.775,E2 26413.775} C_VEL
LIN {X 0,Y 545.506,Z 632.717,A -85,B 0,C 180,E1 26410.595,E2 26410.595} C_VEL
LIN {X 0,Y 545.496,Z 632.715,A -85,B 0,C 180,E1 26407.222,E2 26407.222} C_VEL
LIN {X 0,Y 545.556,Z 632.713,A -85,B 0,C 180,E1 26406.262,E2 26406.262} C_VEL
LIN {X 0,Y 544.597,Z 632.827,A -85,B 0,C 180,E1 26405.453,E2 26405.453} C_VEL
LIN {X 0,Y 538.149,Z 633.634,A -85,B 0,C 180,E1 26403.181,E2 26403.181} C_VEL
LIN {X 0,Y 537.624,Z 633.698,A -85,B 0,C 180,E1 26402.589,E2 26402.589} C_VEL
LIN {X 0,Y 537.623,Z 633.698,A -85,B 0,C 180,E1 26399.163,E2 26399.163} C_VEL
LIN {X 0,Y 537.615,Z 633.696,A -85,B 0,C 180,E1 26395.8,E2 26395.8} C_VEL
LIN {X 0,Y 537.546,Z 633.703,A -85,B 0,C 180,E1 26392.532,E2 26392.532} C_VEL
LIN {X 0,Y 537.576,Z 633.701,A -85,B 0,C 180,E1 26389.11,E2 26389.11} C_VEL
LIN {X 0,Y 537.628,Z 633.701,A -85,B 0,C 180,E1 26385.868,E2 26385.868} C_VEL
LIN {X 0,Y 537.62,Z 633.695,A -85,B 0,C 180,E1 26382.46,E2 26382.46} C_VEL
LIN {X 0,Y 537.628,Z 633.695,A -85,B 0,C 180,E1 26378.989,E2 26378.989} C_VEL
LIN {X 0,Y 537.566,Z 633.704,A -85,B 0,C 180,E1 26375.766,E2 26375.766} C_VEL
LIN {X 0,Y 537.545,Z 633.696,A -85,B 0,C 180,E1 26372.24,E2 26372.24} C_VEL
LIN {X 0,Y 537.626,Z 633.698,A -85,B 0,C 180,E1 26369.042,E2 26369.042} C_VEL
LIN {X 0,Y 537.619,Z 633.69,A -85,B 0,C 180,E1 26365.628,E2 26365.628} C_VEL
LIN {X 0,Y 537.628,Z 633.701,A -85,B 0,C 180,E1 26362.199,E2 26362.199} C_VEL
LIN {X 0,Y 537.604,Z 633.687,A -85,B 0,C 180,E1 26358.849,E2 26358.849} C_VEL
LIN {X 0,Y 537.542,Z 633.705,A -85,B 0,C 180,E1 26355.568,E2 26355.568} C_VEL
LIN {X 0,Y 537.593,Z 633.7,A -85,B 0,C 180,E1 26352.218,E2 26352.218} C_VEL
LIN {X 0,Y 537.626,Z 633.701,A -85,B 0,C 180,E1 26348.966,E2 26348.966} C_VEL
LIN {X 0,Y 537.621,Z 633.702,A -85,B 0,C 180,E1 26345.499,E2 26345.499} C_VEL
LIN {X 0,Y 537.635,Z 633.699,A -85,B 0,C 180,E1 26342.048,E2 26342.048} C_VEL
LIN {X 0,Y 537.554,Z 633.706,A -85,B 0,C 180,E1 26338.823,E2 26338.823} C_VEL
LIN {X 0,Y 537.559,Z 633.705,A -85,B 0,C 180,E1 26335.294,E2 26335.294} C_VEL
LIN {X 0,Y 537.628,Z 633.698,A -85,B 0,C 180,E1 26332.007,E2 26332.007} C_VEL
LIN {X 0,Y 537.621,Z 633.7,A -85,B 0,C 180,E1 26328.542,E2 26328.542} C_VEL
LIN {X 0,Y 537.618,Z 633.697,A -85,B 0,C 180,E1 26325.117,E2 26325.117} C_VEL
LIN {X 0,Y 537.661,Z 633.941,A -85,B 0,C 180,E1 26323.549,E2 26323.549} C_VEL
LIN {X 0,Y 544.832,Z 659.321,A -85,B 0,C 180,E1 26321.121,E2 26321.121} C_VEL
LIN {X 0,Y 546.733,Z 666.951,A -85,B 0,C 180,E1 26320.411,E2 26320.411} C_VEL
LIN {X 0,Y 545.509,Z 711.903,A -85,B 0,C 180,E1 26316.821,E2 26316.821} C_VEL
LIN {X 0,Y 544.375,Z 753.642,A -85,B 0,C 180,E1 26313.503,E2 26313.503} C_VEL
LIN {X 0,Y 543.216,Z 793.673,A -85,B 0,C 180,E1 26310.317,E2 26310.317} C_VEL
LIN {X 0,Y 542.26,Z 832.411,A -85,B 0,C 180,E1 26307.272,E2 26307.272} C_VEL
LIN {X 0,Y 542.47,Z 841.109,A -85,B 0,C 180,E1 26307.128,E2 26307.128} C_VEL
LIN {X 0,Y 540.755,Z 975.835,A -85,B 0,C 180,E1 26305.074,E2 26305.074} C_VEL
LIN {X 0,Y 540.583,Z 992.308,A -85,B 0,C 180,E1 26304.625,E2 26304.625} C_VEL
LIN {X 0,Y 540.272,Z 1007.591,A -85,B 0,C 180,E1 26304.023,E2 26304.023} C_VEL
LIN {X 0,Y 539.858,Z 1022.515,A -85,B 0,C 180,E1 26303.232,E2 26303.232} C_VEL
LIN {X 0,Y 539.39,Z 1036.628,A -85,B 0,C 180,E1 26302.274,E2 26302.274} C_VEL
LIN {X 0,Y 538.86,Z 1049.69,A -85,B 0,C 180,E1 26301.153,E2 26301.153} C_VEL
LIN {X 0,Y 538.357,Z 1061.739,A -85,B 0,C 180,E1 26299.867,E2 26299.867} C_VEL
LIN {X 0,Y 537.876,Z 1072.452,A -85,B 0,C 180,E1 26298.42,E2 26298.42} C_VEL
LIN {X 0,Y 537.527,Z 1080.936,A -85,B 0,C 180,E1 26296.978,E2 26296.978} C_VEL
LIN {X 0,Y 537.249,Z 1088.37,A -85,B 0,C 180,E1 26295.321,E2 26295.321} C_VEL
LIN {X 0,Y 537.097,Z 1093.449,A -85,B 0,C 180,E1 26293.783,E2 26293.783} C_VEL
LIN {X 0,Y 537.005,Z 1097.219,A -85,B 0,C 180,E1 26292.034,E2 26292.034} C_VEL
LIN {X 0,Y 537.013,Z 1099.034,A -85,B 0,C 180,E1 26290.403,E2 26290.403} C_VEL
LIN {X 0,Y 537.098,Z 1099.087,A -85,B 0,C 180,E1 26288.67,E2 26288.67} C_VEL
LIN {X 0,Y 537.268,Z 1097.333,A -85,B 0,C 180,E1 26286.946,E2 26286.946} C_VEL
LIN {X 0,Y 537.541,Z 1093.615,A -85,B 0,C 180,E1 26285.227,E2 26285.227} C_VEL
LIN {X 0,Y 537.911,Z 1088.323,A -85,B 0,C 180,E1 26283.621,E2 26283.621} C_VEL
LIN {X 0,Y 538.394,Z 1080.981,A -85,B 0,C 180,E1 26282.02,E2 26282.02} C_VEL
LIN {X 0,Y 538.949,Z 1072.645,A -85,B 0,C 180,E1 26280.617,E2 26280.617} C_VEL
LIN {X 0,Y 539.595,Z 1062.324,A -85,B 0,C 180,E1 26279.254,E2 26279.254} C_VEL
LIN {X 0,Y 540.258,Z 1050.84,A -85,B 0,C 180,E1 26278.036,E2 26278.036} C_VEL
LIN {X 0,Y 540.94,Z 1036.96,A -85,B 0,C 180,E1 26276.872,E2 26276.872} C_VEL
LIN {X 0,Y 541.452,Z 1023.323,A -85,B 0,C 180,E1 26275.974,E2 26275.974} C_VEL
LIN {X 0,Y 541.854,Z 1009.819,A -85,B 0,C 180,E1 26275.288,E2 26275.288} C_VEL
LIN {X 0,Y 542.144,Z 996.496,A -85,B 0,C 180,E1 26274.766,E2 26274.766} C_VEL
LIN {X 0,Y 542.311,Z 981.575,A -85,B 0,C 180,E1 26274.337,E2 26274.337} C_VEL
LIN {X 0,Y 542.711,Z 938.612,A -85,B 0,C 180,E1 26273.631,E2 26273.631} C_VEL
LIN {X 0,Y 544.853,Z 839.61,A -85,B 0,C 180,E1 26272.007,E2 26272.007} C_VEL
LIN {X 0,Y 545.362,Z 831.79,A -85,B 0,C 180,E1 26271.404,E2 26271.404} C_VEL
LIN {X 0,Y 546.673,Z 787.093,A -85,B 0,C 180,E1 26267.909,E2 26267.909} C_VEL
LIN {X 0,Y 547.794,Z 742.784,A -85,B 0,C 180,E1 26264.493,E2 26264.493} C_VEL
LIN {X 0,Y 548.759,Z 699.797,A -85,B 0,C 180,E1 26261.238,E2 26261.238} C_VEL
LIN {X 0,Y 549.427,Z 667.417,A -85,B 0,C 180,E1 26258.821,E2 26258.821} C_VEL
LIN {X 0,Y 544.578,Z 651.526,A -85,B 0,C 180,E1 26257.256,E2 26257.256} C_VEL
LIN {X 0,Y 538.717,Z 636.875,A -85,B 0,C 180,E1 26255.665,E2 26255.665} C_VEL
LIN {X 0,Y 537.594,Z 633.712,A -85,B 0,C 180,E1 26255.318,E2 26255.318} C_VEL
LIN {X 0,Y 537.604,Z 633.706,A -85,B 0,C 180,E1 26252.048,E2 26252.048} C_VEL
LIN {X 0,Y 537.619,Z 633.703,A -85,B 0,C 180,E1 26248.74,E2 26248.74} C_VEL
LIN {X 0,Y 537.622,Z 633.699,A -85,B 0,C 180,E1 26245.1,E2 26245.1} C_VEL
LIN {X 0,Y 537.633,Z 633.699,A -85,B 0,C 180,E1 26241.596,E2 26241.596} C_VEL
LIN {X 0,Y 537.597,Z 633.703,A -85,B 0,C 180,E1 26238.107,E2 26238.107} C_VEL
LIN {X 0,Y 537.61,Z 633.697,A -85,B 0,C 180,E1 26234.818,E2 26234.818} C_VEL
LIN {X 0,Y 537.626,Z 633.809,A -85,B 0,C 180,E1 26231.508,E2 26231.508} C_VEL
LIN {X 0,Y 545.819,Z 658.606,A -85,B 0,C 180,E1 26228.195,E2 26228.195} C_VEL
LIN {X 0,Y 552.025,Z 678.213,A -85,B 0,C 180,E1 26225.772,E2 26225.772} C_VEL
LIN {X 0,Y 555.424,Z 685.912,A -85,B 0,C 180,E1 26225.405,E2 26225.405} C_VEL
LIN {X 0,Y 562.595,Z 723.543,A -85,B 0,C 180,E1 26224.278,E2 26224.278} C_VEL
LIN {X 0,Y 555.798,Z 955.584,A -85,B 0,C 180,E1 26220.74,E2 26220.74} C_VEL
LIN {X 0,Y 554.753,Z 987.349,A -85,B 0,C 180,E1 26220.215,E2 26220.215} C_VEL
LIN {X 0,Y 553.554,Z 1009.512,A -85,B 0,C 180,E1 26219.674,E2 26219.674} C_VEL
LIN {X 0,Y 552.062,Z 1031.137,A -85,B 0,C 180,E1 26218.955,E2 26218.955} C_VEL
LIN {X 0,Y 550.39,Z 1052.177,A -85,B 0,C 180,E1 26218.066,E2 26218.066} C_VEL
LIN {X 0,Y 548.57,Z 1072.948,A -85,B 0,C 180,E1 26216.989,E2 26216.989} C_VEL
LIN {X 0,Y 546.715,Z 1092.504,A -85,B 0,C 180,E1 26215.772,E2 26215.772} C_VEL
LIN {X 0,Y 544.841,Z 1111.123,A -85,B 0,C 180,E1 26214.386,E2 26214.386} C_VEL
LIN {X 0,Y 542.989,Z 1129.239,A -85,B 0,C 180,E1 26212.805,E2 26212.805} C_VEL
LIN {X 0,Y 541.304,Z 1145.832,A -85,B 0,C 180,E1 26211.111,E2 26211.111} C_VEL
LIN {X 0,Y 539.883,Z 1160.515,A -85,B 0,C 180,E1 26209.359,E2 26209.359} C_VEL
LIN {X 0,Y 538.656,Z 1173.819,A -85,B 0,C 180,E1 26207.499,E2 26207.499} C_VEL
LIN {X 0,Y 537.628,Z 1186.491,A -85,B 0,C 180,E1 26205.422,E2 26205.422} C_VEL
LIN {X 0,Y 536.906,Z 1197.146,A -85,B 0,C 180,E1 26203.35,E2 26203.35} C_VEL
LIN {X 0,Y 536.408,Z 1206.254,A -85,B 0,C 180,E1 26201.177,E2 26201.177} C_VEL
LIN {X 0,Y 536.125,Z 1213.896,A -85,B 0,C 180,E1 26198.903,E2 26198.903} C_VEL
LIN {X 0,Y 535.996,Z 1219.506,A -85,B 0,C 180,E1 26196.748,E2 26196.748} C_VEL
LIN {X 0,Y 535.973,Z 1223.396,A -85,B 0,C 180,E1 26194.6,E2 26194.6} C_VEL
LIN {X 0,Y 535.99,Z 1225.974,A -85,B 0,C 180,E1 26192.244,E2 26192.244} C_VEL
LIN {X 0,Y 536.006,Z 1226.793,A -85,B 0,C 180,E1 26189.999,E2 26189.999} C_VEL
LIN {X 0,Y 535.998,Z 1225.836,A -85,B 0,C 180,E1 26187.753,E2 26187.753} C_VEL
LIN {X 0,Y 535.983,Z 1223.118,A -85,B 0,C 180,E1 26185.398,E2 26185.398} C_VEL
LIN {X 0,Y 536.006,Z 1219.058,A -85,B 0,C 180,E1 26183.249,E2 26183.249} C_VEL
LIN {X 0,Y 536.129,Z 1213.286,A -85,B 0,C 180,E1 26181.094,E2 26181.094} C_VEL
LIN {X 0,Y 536.386,Z 1205.865,A -85,B 0,C 180,E1 26178.929,E2 26178.929} C_VEL
LIN {X 0,Y 536.847,Z 1196.551,A -85,B 0,C 180,E1 26176.755,E2 26176.755} C_VEL
LIN {X 0,Y 537.522,Z 1185.726,A -85,B 0,C 180,E1 26174.683,E2 26174.683} C_VEL
LIN {X 0,Y 538.491,Z 1172.84,A -85,B 0,C 180,E1 26172.604,E2 26172.604} C_VEL
LIN {X 0,Y 539.653,Z 1159.278,A -85,B 0,C 180,E1 26170.742,E2 26170.742} C_VEL
LIN {X 0,Y 541.016,Z 1144.017,A -85,B 0,C 180,E1 26168.962,E2 26168.962} C_VEL
LIN {X 0,Y 542.66,Z 1126.767,A -85,B 0,C 180,E1 26167.235,E2 26167.235} C_VEL
LIN {X 0,Y 544.391,Z 1108.932,A -85,B 0,C 180,E1 26165.705,E2 26165.705} C_VEL
LIN {X 0,Y 546.239,Z 1089.561,A -85,B 0,C 180,E1 26164.288,E2 26164.288} C_VEL
LIN {X 0,Y 548.102,Z 1069.214,A -85,B 0,C 180,E1 26163.041,E2 26163.041} C_VEL
LIN {X 0,Y 549.944,Z 1047.824,A -85,B 0,C 180,E1 26161.948,E2 26161.948} C_VEL
LIN {X 0,Y 551.74,Z 1025.861,A -85,B 0,C 180,E1 26161.031,E2 26161.031} C_VEL
LIN {X 0,Y 553.374,Z 1003.208,A -85,B 0,C 180,E1 26160.279,E2 26160.279} C_VEL
LIN {X 0,Y 554.937,Z 978.037,A -85,B 0,C 180,E1 26159.667,E2 26159.667} C_VEL
LIN {X 0,Y 559.423,Z 869.198,A -85,B 0,C 180,E1 26157.747,E2 26157.747} C_VEL
LIN {X 0,Y 564.722,Z 778.809,A -85,B 0,C 180,E1 26156.008,E2 26156.008} C_VEL
LIN {X 0,Y 568.713,Z 722.948,A -85,B 0,C 180,E1 26154.853,E2 26154.853} C_VEL
LIN {X 0,Y 566.411,Z 700.432,A -85,B 0,C 180,E1 26153.883,E2 26153.883} C_VEL
LIN {X 0,Y 565.152,Z 691.839,A -85,B 0,C 180,E1 26153.423,E2 26153.423} C_VEL
LIN {X 0,Y 561.069,Z 682.635,A -85,B 0,C 180,E1 26152.515,E2 26152.515} C_VEL
LIN {X 0,Y 557.983,Z 676.368,A -85,B 0,C 180,E1 26151.753,E2 26151.753} C_VEL
LIN {X 0,Y 554.243,Z 669.243,A -85,B 0,C 180,E1 26150.71,E2 26150.71} C_VEL
LIN {X 0,Y 549.739,Z 661.281,A -85,B 0,C 180,E1 26149.171,E2 26149.171} C_VEL
LIN {X 0,Y 548.431,Z 657.778,A -85,B 0,C 180,E1 26148.001,E2 26148.001} C_VEL
LIN {X 0,Y 547.456,Z 655.176,A -85,B 0,C 180,E1 26146.914,E2 26146.914} C_VEL
LIN {X 0,Y 546.271,Z 651.869,A -85,B 0,C 180,E1 26144.748,E2 26144.748} C_VEL
LIN {X 0,Y 545.803,Z 651.288,A -85,B 0,C 180,E1 26142.676,E2 26142.676} C_VEL
LIN {X 0,Y 546.159,Z 651.707,A -85,B 0,C 180,E1 26141.986,E2 26141.986} C_VEL
LIN {X 0,Y 548.574,Z 654.276,A -85,B 0,C 180,E1 26140.689,E2 26140.689} C_VEL
LIN {X 0,Y 552.221,Z 658.359,A -85,B 0,C 180,E1 26139.328,E2 26139.328} C_VEL
LIN {X 0,Y 554.275,Z 660.807,A -85,B 0,C 180,E1 26138.719,E2 26138.719} C_VEL
LIN {X 0,Y 557.838,Z 665.481,A -85,B 0,C 180,E1 26137.77,E2 26137.77} C_VEL
LIN {X 0,Y 561.142,Z 670.254,A -85,B 0,C 180,E1 26136.99,E2 26136.99} C_VEL
LIN {X 0,Y 565.759,Z 677.409,A -85,B 0,C 180,E1 26136.029,E2 26136.029} C_VEL
LIN {X 0,Y 570.832,Z 686.629,A -85,B 0,C 180,E1 26135.069,E2 26135.069} C_VEL
LIN {X 0,Y 564.142,Z 772.655,A -85,B 0,C 180,E1 26133.304,E2 26133.304} C_VEL
LIN {X 0,Y 559.316,Z 855.75,A -85,B 0,C 180,E1 26131.716,E2 26131.716} C_VEL
LIN {X 0,Y 555.65,Z 941.184,A -85,B 0,C 180,E1 26130.175,E2 26130.175} C_VEL
LIN {X 0,Y 554.467,Z 964.414,A -85,B 0,C 180,E1 26129.561,E2 26129.561} C_VEL
LIN {X 0,Y 553.012,Z 986.304,A -85,B 0,C 180,E1 26128.789,E2 26128.789} C_VEL
LIN {X 0,Y 551.387,Z 1007.267,A -85,B 0,C 180,E1 26127.855,E2 26127.855} C_VEL
LIN {X 0,Y 549.55,Z 1028.348,A -85,B 0,C 180,E1 26126.708,E2 26126.708} C_VEL
LIN {X 0,Y 547.726,Z 1047.429,A -85,B 0,C 180,E1 26125.462,E2 26125.462} C_VEL
LIN {X 0,Y 545.805,Z 1066.309,A -85,B 0,C 180,E1 26123.999,E2 26123.999} C_VEL
LIN {X 0,Y 543.943,Z 1083.412,A -85,B 0,C 180,E1 26122.424,E2 26122.424} C_VEL
LIN {X 0,Y 542.228,Z 1099.062,A -85,B 0,C 180,E1 26120.738,E2 26120.738} C_VEL
LIN {X 0,Y 540.743,Z 1112.987,A -85,B 0,C 180,E1 26118.994,E2 26118.994} C_VEL
LIN {X 0,Y 539.364,Z 1126.284,A -85,B 0,C 180,E1 26117.034,E2 26117.034} C_VEL
LIN {X 0,Y 538.27,Z 1137.439,A -85,B 0,C 180,E1 26115.076,E2 26115.076} C_VEL
LIN {X 0,Y 537.393,Z 1147.822,A -85,B 0,C 180,E1 26112.904,E2 26112.904} C_VEL
LIN {X 0,Y 536.785,Z 1156.31,A -85,B 0,C 180,E1 26110.738,E2 26110.738} C_VEL
LIN {X 0,Y 536.39,Z 1162.919,A -85,B 0,C 180,E1 26108.579,E2 26108.579} C_VEL
LIN {X 0,Y 536.151,Z 1168.381,A -85,B 0,C 180,E1 26106.212,E2 26106.212} C_VEL
LIN {X 0,Y 536.045,Z 1171.943,A -85,B 0,C 180,E1 26103.96,E2 26103.96} C_VEL
LIN {X 0,Y 536.011,Z 1173.819,A -85,B 0,C 180,E1 26101.713,E2 26101.713} C_VEL
LIN {X 0,Y 536.006,Z 1174.118,A -85,B 0,C 180,E1 26099.361,E2 26099.361} C_VEL
LIN {X 0,Y 536.016,Z 1172.864,A -85,B 0,C 180,E1 26097.115,E2 26097.115} C_VEL
LIN {X 0,Y 536.065,Z 1169.945,A -85,B 0,C 180,E1 26094.866,E2 26094.866} C_VEL
LIN {X 0,Y 536.2,Z 1165.412,A -85,B 0,C 180,E1 26092.61,E2 26092.61} C_VEL
LIN {X 0,Y 536.481,Z 1159.214,A -85,B 0,C 180,E1 26090.346,E2 26090.346} C_VEL
LIN {X 0,Y 536.927,Z 1151.522,A -85,B 0,C 180,E1 26088.182,E2 26088.182} C_VEL
LIN {X 0,Y 537.611,Z 1141.985,A -85,B 0,C 180,E1 26086.011,E2 26086.011} C_VEL
LIN {X 0,Y 538.552,Z 1131.068,A -85,B 0,C 180,E1 26083.943,E2 26083.943} C_VEL
LIN {X 0,Y 539.733,Z 1118.759,A -85,B 0,C 180,E1 26081.981,E2 26081.981} C_VEL
LIN {X 0,Y 541.118,Z 1105.013,A -85,B 0,C 180,E1 26080.126,E2 26080.126} C_VEL
LIN {X 0,Y 542.811,Z 1088.909,A -85,B 0,C 180,E1 26078.272,E2 26078.272} C_VEL
LIN {X 0,Y 544.58,Z 1072.284,A -85,B 0,C 180,E1 26076.638,E2 26076.638} C_VEL
LIN {X 0,Y 546.366,Z 1055,A -85,B 0,C 180,E1 26075.193,E2 26075.193} C_VEL
LIN {X 0,Y 548.194,Z 1036.357,A -85,B 0,C 180,E1 26073.868,E2 26073.868} C_VEL
LIN {X 0,Y 549.996,Z 1016.526,A -85,B 0,C 180,E1 26072.678,E2 26072.678} C_VEL
LIN {X 0,Y 551.715,Z 995.943,A -85,B 0,C 180,E1 26071.655,E2 26071.655} C_VEL
LIN {X 0,Y 553.221,Z 974.2,A -85,B 0,C 180,E1 26070.794,E2 26070.794} C_VEL
LIN {X 0,Y 554.488,Z 952.142,A -85,B 0,C 180,E1 26070.118,E2 26070.118} C_VEL
LIN {X 0,Y 555.481,Z 929.585,A -85,B 0,C 180,E1 26069.616,E2 26069.616} C_VEL
LIN {X 0,Y 562.807,Z 681.039,A -85,B 0,C 180,E1 26065.824,E2 26065.824} C_VEL
LIN {X 0,Y 553.23,Z 662.152,A -85,B 0,C 180,E1 26064.87,E2 26064.87} C_VEL
LIN {X 0,Y 538.901,Z 637.212,A -85,B 0,C 180,E1 26063.435,E2 26063.435} C_VEL
LIN {X 0,Y 537.59,Z 633.703,A -85,B 0,C 180,E1 26063.246,E2 26063.246} C_VEL
LIN {X 0,Y 537.604,Z 633.698,A -85,B 0,C 180,E1 26059.856,E2 26059.856} C_VEL
LIN {X 0,Y 537.615,Z 633.697,A -85,B 0,C 180,E1 26056.499,E2 26056.499} C_VEL
LIN {X 0,Y 537.58,Z 633.704,A -85,B 0,C 180,E1 26053.193,E2 26053.193} C_VEL
LIN {X 0,Y 537.598,Z 633.703,A -85,B 0,C 180,E1 26049.918,E2 26049.918} C_VEL
LIN {X 0,Y 537.58,Z 633.705,A -85,B 0,C 180,E1 26046.66,E2 26046.66} C_VEL
LIN {X 0,Y 537.595,Z 633.701,A -85,B 0,C 180,E1 26043.278,E2 26043.278} C_VEL
LIN {X 0,Y 537.624,Z 633.698,A -85,B 0,C 180,E1 26042.589,E2 26042.589} C_VEL
LIN {X 0,Y 536.656,Z 633.82,A -85,B 0,C 180,E1 26041.768,E2 26041.768} C_VEL
LIN {X 0,Y 530.138,Z 634.629,A -85,B 0,C 180,E1 26039.403,E2 26039.403} C_VEL
LIN {X 0,Y 529.686,Z 634.689,A -85,B 0,C 180,E1 26038.862,E2 26038.862} C_VEL
LIN {X 0,Y 529.685,Z 634.687,A -85,B 0,C 180,E1 26035.374,E2 26035.374} C_VEL
LIN {X 0,Y 529.623,Z 634.691,A -85,B 0,C 180,E1 26032.069,E2 26032.069} C_VEL
LIN {X 0,Y 529.624,Z 634.69,A -85,B 0,C 180,E1 26028.721,E2 26028.721} C_VEL
LIN {X 0,Y 529.688,Z 634.685,A -85,B 0,C 180,E1 26025.437,E2 26025.437} C_VEL
LIN {X 0,Y 529.675,Z 634.69,A -85,B 0,C 180,E1 26021.986,E2 26021.986} C_VEL
LIN {X 0,Y 529.673,Z 634.682,A -85,B 0,C 180,E1 26018.578,E2 26018.578} C_VEL
LIN {X 0,Y 529.658,Z 634.692,A -85,B 0,C 180,E1 26015.309,E2 26015.309} C_VEL
LIN {X 0,Y 529.61,Z 634.685,A -85,B 0,C 180,E1 26011.949,E2 26011.949} C_VEL
LIN {X 0,Y 529.65,Z 634.688,A -85,B 0,C 180,E1 26008.487,E2 26008.487} C_VEL
LIN {X 0,Y 529.682,Z 634.679,A -85,B 0,C 180,E1 26005.129,E2 26005.129} C_VEL
LIN {X 0,Y 529.661,Z 634.688,A -85,B 0,C 180,E1 26001.644,E2 26001.644} C_VEL
LIN {X 0,Y 529.661,Z 634.678,A -85,B 0,C 180,E1 25998.238,E2 25998.238} C_VEL
LIN {X 0,Y 529.64,Z 634.694,A -85,B 0,C 180,E1 25994.901,E2 25994.901} C_VEL
LIN {X 0,Y 529.636,Z 634.691,A -85,B 0,C 180,E1 25991.624,E2 25991.624} C_VEL
LIN {X 0,Y 529.677,Z 634.686,A -85,B 0,C 180,E1 25988.17,E2 25988.17} C_VEL
LIN {X 0,Y 529.667,Z 634.688,A -85,B 0,C 180,E1 25984.867,E2 25984.867} C_VEL
LIN {X 0,Y 529.654,Z 634.694,A -85,B 0,C 180,E1 25981.472,E2 25981.472} C_VEL
LIN {X 0,Y 529.669,Z 634.693,A -85,B 0,C 180,E1 25978.15,E2 25978.15} C_VEL
LIN {X 0,Y 529.639,Z 634.695,A -85,B 0,C 180,E1 25974.714,E2 25974.714} C_VEL
LIN {X 0,Y 529.656,Z 634.69,A -85,B 0,C 180,E1 25971.33,E2 25971.33} C_VEL
LIN {X 0,Y 529.685,Z 634.686,A -85,B 0,C 180,E1 25967.925,E2 25967.925} C_VEL
LIN {X 0,Y 529.649,Z 634.692,A -85,B 0,C 180,E1 25964.474,E2 25964.474} C_VEL
LIN {X 0,Y 529.677,Z 634.739,A -85,B 0,C 180,E1 25963.886,E2 25963.886} C_VEL
LIN {X 0,Y 537.409,Z 662.005,A -85,B 0,C 180,E1 25961.268,E2 25961.268} C_VEL
LIN {X 0,Y 539.187,Z 669.007,A -85,B 0,C 180,E1 25960.606,E2 25960.606} C_VEL
LIN {X 0,Y 537.882,Z 714.632,A -85,B 0,C 180,E1 25956.936,E2 25956.936} C_VEL
LIN {X 0,Y 536.623,Z 757.029,A -85,B 0,C 180,E1 25953.533,E2 25953.533} C_VEL
LIN {X 0,Y 535.474,Z 797.03,A -85,B 0,C 180,E1 25950.341,E2 25950.341} C_VEL
LIN {X 0,Y 534.532,Z 833.126,A -85,B 0,C 180,E1 25947.483,E2 25947.483} C_VEL
LIN {X 0,Y 534.72,Z 842.376,A -85,B 0,C 180,E1 25947.329,E2 25947.329} C_VEL
LIN {X 0,Y 532.927,Z 976.404,A -85,B 0,C 180,E1 25945.243,E2 25945.243} C_VEL
LIN {X 0,Y 532.756,Z 992.622,A -85,B 0,C 180,E1 25944.798,E2 25944.798} C_VEL
LIN {X 0,Y 532.422,Z 1008.551,A -85,B 0,C 180,E1 25944.164,E2 25944.164} C_VEL
LIN {X 0,Y 531.995,Z 1023.456,A -85,B 0,C 180,E1 25943.361,E2 25943.361} C_VEL
LIN {X 0,Y 531.509,Z 1037.573,A -85,B 0,C 180,E1 25942.389,E2 25942.389} C_VEL
LIN {X 0,Y 530.953,Z 1050.867,A -85,B 0,C 180,E1 25941.229,E2 25941.229} C_VEL
LIN {X 0,Y 530.443,Z 1062.695,A -85,B 0,C 180,E1 25939.946,E2 25939.946} C_VEL
LIN {X 0,Y 529.946,Z 1073.416,A -85,B 0,C 180,E1 25938.477,E2 25938.477} C_VEL
LIN {X 0,Y 529.586,Z 1081.907,A -85,B 0,C 180,E1 25937.014,E2 25937.014} C_VEL
LIN {X 0,Y 529.302,Z 1089.346,A -85,B 0,C 180,E1 25935.333,E2 25935.333} C_VEL
LIN {X 0,Y 529.146,Z 1094.429,A -85,B 0,C 180,E1 25933.771,E2 25933.771} C_VEL
LIN {X 0,Y 529.055,Z 1098.202,A -85,B 0,C 180,E1 25931.996,E2 25931.996} C_VEL
LIN {X 0,Y 529.071,Z 1100.014,A -85,B 0,C 180,E1 25930.34,E2 25930.34} C_VEL
LIN {X 0,Y 529.168,Z 1100.058,A -85,B 0,C 180,E1 25928.582,E2 25928.582} C_VEL
LIN {X 0,Y 529.344,Z 1098.453,A -85,B 0,C 180,E1 25926.941,E2 25926.941} C_VEL
LIN {X 0,Y 529.612,Z 1095.11,A -85,B 0,C 180,E1 25925.306,E2 25925.306} C_VEL
LIN {X 0,Y 530.001,Z 1089.964,A -85,B 0,C 180,E1 25923.662,E2 25923.662} C_VEL
LIN {X 0,Y 530.47,Z 1083.459,A -85,B 0,C 180,E1 25922.158,E2 25922.158} C_VEL
LIN {X 0,Y 531.075,Z 1074.939,A -85,B 0,C 180,E1 25920.645,E2 25920.645} C_VEL
LIN {X 0,Y 531.714,Z 1065.745,A -85,B 0,C 180,E1 25919.351,E2 25919.351} C_VEL
LIN {X 0,Y 532.454,Z 1053.705,A -85,B 0,C 180,E1 25918.007,E2 25918.007} C_VEL
LIN {X 0,Y 533.148,Z 1040.995,A -85,B 0,C 180,E1 25916.88,E2 25916.88} C_VEL
LIN {X 0,Y 533.758,Z 1026.434,A -85,B 0,C 180,E1 25915.862,E2 25915.862} C_VEL
LIN {X 0,Y 534.219,Z 1012.421,A -85,B 0,C 180,E1 25915.112,E2 25915.112} C_VEL
LIN {X 0,Y 534.554,Z 997.96,A -85,B 0,C 180,E1 25914.53,E2 25914.53} C_VEL
LIN {X 0,Y 534.737,Z 982.681,A -85,B 0,C 180,E1 25914.081,E2 25914.081} C_VEL
LIN {X 0,Y 535.128,Z 942.597,A -85,B 0,C 180,E1 25913.401,E2 25913.401} C_VEL
LIN {X 0,Y 537.509,Z 840.735,A -85,B 0,C 180,E1 25911.682,E2 25911.682} C_VEL
LIN {X 0,Y 538.004,Z 833.477,A -85,B 0,C 180,E1 25911.124,E2 25911.124} C_VEL
LIN {X 0,Y 539.262,Z 792.599,A -85,B 0,C 180,E1 25907.904,E2 25907.904} C_VEL
LIN {X 0,Y 540.511,Z 748.727,A -85,B 0,C 180,E1 25904.494,E2 25904.494} C_VEL
LIN {X 0,Y 541.513,Z 710.116,A -85,B 0,C 180,E1 25901.536,E2 25901.536} C_VEL
LIN {X 0,Y 542.482,Z 670.55,A -85,B 0,C 180,E1 25898.554,E2 25898.554} C_VEL
LIN {X 0,Y 537.737,Z 654.957,A -85,B 0,C 180,E1 25896.982,E2 25896.982} C_VEL
LIN {X 0,Y 532.147,Z 641.021,A -85,B 0,C 180,E1 25895.42,E2 25895.42} C_VEL
LIN {X 0,Y 529.684,Z 634.88,A -85,B 0,C 180,E1 25894.712,E2 25894.712} C_VEL
LIN {X 0,Y 529.674,Z 634.691,A -85,B 0,C 180,E1 25891.469,E2 25891.469} C_VEL
LIN {X 0,Y 529.66,Z 634.692,A -85,B 0,C 180,E1 25888.216,E2 25888.216} C_VEL
LIN {X 0,Y 529.684,Z 634.689,A -85,B 0,C 180,E1 25884.713,E2 25884.713} C_VEL
LIN {X 0,Y 529.683,Z 634.69,A -85,B 0,C 180,E1 25881.189,E2 25881.189} C_VEL
LIN {X 0,Y 529.686,Z 634.691,A -85,B 0,C 180,E1 25877.726,E2 25877.726} C_VEL
LIN {X 0,Y 529.649,Z 634.688,A -85,B 0,C 180,E1 25874.304,E2 25874.304} C_VEL
LIN {X 0,Y 529.707,Z 634.912,A -85,B 0,C 180,E1 25872.002,E2 25872.002} C_VEL
LIN {X 0,Y 537.691,Z 658.924,A -85,B 0,C 180,E1 25868.728,E2 25868.728} C_VEL
LIN {X 0,Y 543.736,Z 677.92,A -85,B 0,C 180,E1 25866.333,E2 25866.333} C_VEL
LIN {X 0,Y 548.953,Z 689.065,A -85,B 0,C 180,E1 25865.778,E2 25865.778} C_VEL
LIN {X 0,Y 555.72,Z 724.89,A -85,B 0,C 180,E1 25864.686,E2 25864.686} C_VEL
LIN {X 0,Y 549.024,Z 939.531,A -85,B 0,C 180,E1 25861.347,E2 25861.347} C_VEL
LIN {X 0,Y 547.602,Z 984.928,A -85,B 0,C 180,E1 25860.614,E2 25860.614} C_VEL
LIN {X 0,Y 546.335,Z 1007.78,A -85,B 0,C 180,E1 25860.061,E2 25860.061} C_VEL
LIN {X 0,Y 544.77,Z 1029.918,A -85,B 0,C 180,E1 25859.325,E2 25859.325} C_VEL
LIN {X 0,Y 543.014,Z 1051.261,A -85,B 0,C 180,E1 25858.422,E2 25858.422} C_VEL
LIN {X 0,Y 541.221,Z 1071.241,A -85,B 0,C 180,E1 25857.386,E2 25857.386} C_VEL
LIN {X 0,Y 539.229,Z 1091.368,A -85,B 0,C 180,E1 25856.127,E2 25856.127} C_VEL
LIN {X 0,Y 537.318,Z 1109.814,A -85,B 0,C 180,E1 25854.751,E2 25854.751} C_VEL
LIN {X 0,Y 535.358,Z 1128.152,A -85,B 0,C 180,E1 25853.143,E2 25853.143} C_VEL
LIN {X 0,Y 533.66,Z 1144.345,A -85,B 0,C 180,E1 25851.486,E2 25851.486} C_VEL
LIN {X 0,Y 532.105,Z 1159.592,A -85,B 0,C 180,E1 25849.654,E2 25849.654} C_VEL
LIN {X 0,Y 530.812,Z 1173.027,A -85,B 0,C 180,E1 25847.766,E2 25847.766} C_VEL
LIN {X 0,Y 529.754,Z 1185.505,A -85,B 0,C 180,E1 25845.714,E2 25845.714} C_VEL
LIN {X 0,Y 528.995,Z 1195.984,A -85,B 0,C 180,E1 25843.665,E2 25843.665} C_VEL
LIN {X 0,Y 528.472,Z 1204.847,A -85,B 0,C 180,E1 25841.568,E2 25841.568} C_VEL
LIN {X 0,Y 528.164,Z 1212.445,A -85,B 0,C 180,E1 25839.368,E2 25839.368} C_VEL
LIN {X 0,Y 528.024,Z 1218.266,A -85,B 0,C 180,E1 25837.178,E2 25837.178} C_VEL
LIN {X 0,Y 527.975,Z 1222.633,A -85,B 0,C 180,E1 25834.887,E2 25834.887} C_VEL
LIN {X 0,Y 527.988,Z 1225.289,A -85,B 0,C 180,E1 25832.712,E2 25832.712} C_VEL
LIN {X 0,Y 528.001,Z 1226.296,A -85,B 0,C 180,E1 25830.541,E2 25830.541} C_VEL
LIN {X 0,Y 528.002,Z 1225.821,A -85,B 0,C 180,E1 25828.262,E2 25828.262} C_VEL
LIN {X 0,Y 527.996,Z 1223.789,A -85,B 0,C 180,E1 25826.089,E2 25826.089} C_VEL
LIN {X 0,Y 528.008,Z 1219.983,A -85,B 0,C 180,E1 25823.802,E2 25823.802} C_VEL
LIN {X 0,Y 528.1,Z 1214.794,A -85,B 0,C 180,E1 25821.616,E2 25821.616} C_VEL
LIN {X 0,Y 528.309,Z 1207.795,A -85,B 0,C 180,E1 25819.42,E2 25819.42} C_VEL
LIN {X 0,Y 528.725,Z 1199.005,A -85,B 0,C 180,E1 25817.215,E2 25817.215} C_VEL
LIN {X 0,Y 529.365,Z 1188.87,A -85,B 0,C 180,E1 25815.114,E2 25815.114} C_VEL
LIN {X 0,Y 530.291,Z 1176.59,A -85,B 0,C 180,E1 25813.005,E2 25813.005} C_VEL
LIN {X 0,Y 531.407,Z 1163.631,A -85,B 0,C 180,E1 25811.116,E2 25811.116} C_VEL
LIN {X 0,Y 532.839,Z 1148.55,A -85,B 0,C 180,E1 25809.226,E2 25809.226} C_VEL
LIN {X 0,Y 534.507,Z 1131.913,A -85,B 0,C 180,E1 25807.449,E2 25807.449} C_VEL
LIN {X 0,Y 536.256,Z 1114.419,A -85,B 0,C 180,E1 25805.856,E2 25805.856} C_VEL
LIN {X 0,Y 538.31,Z 1094.289,A -85,B 0,C 180,E1 25804.295,E2 25804.295} C_VEL
LIN {X 0,Y 540.298,Z 1074.154,A -85,B 0,C 180,E1 25802.977,E2 25802.977} C_VEL
LIN {X 0,Y 542.274,Z 1053.312,A -85,B 0,C 180,E1 25801.832,E2 25801.832} C_VEL
LIN {X 0,Y 544.165,Z 1031.605,A -85,B 0,C 180,E1 25800.86,E2 25800.86} C_VEL
LIN {X 0,Y 545.97,Z 1009.005,A -85,B 0,C 180,E1 25800.048,E2 25800.048} C_VEL
LIN {X 0,Y 547.659,Z 984.678,A -85,B 0,C 180,E1 25799.384,E2 25799.384} C_VEL
LIN {X 0,Y 549.046,Z 956.642,A -85,B 0,C 180,E1 25798.839,E2 25798.839} C_VEL
LIN {X 0,Y 552.997,Z 870.82,A -85,B 0,C 180,E1 25797.272,E2 25797.272} C_VEL
LIN {X 0,Y 558.524,Z 784.435,A -85,B 0,C 180,E1 25795.555,E2 25795.555} C_VEL
LIN {X 0,Y 563.218,Z 724.658,A -85,B 0,C 180,E1 25794.283,E2 25794.283} C_VEL
LIN {X 0,Y 561.32,Z 702.935,A -85,B 0,C 180,E1 25793.305,E2 25793.305} C_VEL
LIN {X 0,Y 560.359,Z 696.125,A -85,B 0,C 180,E1 25792.926,E2 25792.926} C_VEL
LIN {X 0,Y 556.638,Z 687.458,A -85,B 0,C 180,E1 25792.009,E2 25792.009} C_VEL
LIN {X 0,Y 553.902,Z 681.665,A -85,B 0,C 180,E1 25791.268,E2 25791.268} C_VEL
LIN {X 0,Y 550.95,Z 675.88,A -85,B 0,C 180,E1 25790.392,E2 25790.392} C_VEL
LIN {X 0,Y 547.002,Z 668.369,A -85,B 0,C 180,E1 25788.903,E2 25788.903} C_VEL
LIN {X 0,Y 544.813,Z 664.783,A -85,B 0,C 180,E1 25787.858,E2 25787.858} C_VEL
LIN {X 0,Y 543.413,Z 662.147,A -85,B 0,C 180,E1 25786.929,E2 25786.929} C_VEL
LIN {X 0,Y 542.194,Z 659.384,A -85,B 0,C 180,E1 25785.361,E2 25785.361} C_VEL
LIN {X 0,Y 542.088,Z 658.61,A -85,B 0,C 180,E1 25784.502,E2 25784.502} C_VEL
LIN {X 0,Y 542.849,Z 658.73,A -85,B 0,C 180,E1 25783.008,E2 25783.008} C_VEL
LIN {X 0,Y 544.263,Z 659.612,A -85,B 0,C 180,E1 25781.922,E2 25781.922} C_VEL
LIN {X 0,Y 546.848,Z 662.459,A -85,B 0,C 180,E1 25780.559,E2 25780.559} C_VEL
LIN {X 0,Y 550.999,Z 667.277,A -85,B 0,C 180,E1 25779.082,E2 25779.082} C_VEL
LIN {X 0,Y 554.789,Z 672.588,A -85,B 0,C 180,E1 25777.995,E2 25777.995} C_VEL
LIN {X 0,Y 558.232,Z 677.752,A -85,B 0,C 180,E1 25777.148,E2 25777.148} C_VEL
LIN {X 0,Y 562.859,Z 685.394,A -85,B 0,C 180,E1 25776.143,E2 25776.143} C_VEL
LIN {X 0,Y 565.408,Z 690.565,A -85,B 0,C 180,E1 25775.615,E2 25775.615} C_VEL
LIN {X 0,Y 558.019,Z 777.414,A -85,B 0,C 180,E1 25773.776,E2 25773.776} C_VEL
LIN {X 0,Y 552.713,Z 860.972,A -85,B 0,C 180,E1 25772.126,E2 25772.126} C_VEL
LIN {X 0,Y 548.893,Z 942.194,A -85,B 0,C 180,E1 25770.609,E2 25770.609} C_VEL
LIN {X 0,Y 547.598,Z 965.501,A -85,B 0,C 180,E1 25769.973,E2 25769.973} C_VEL
LIN {X 0,Y 546.071,Z 986.984,A -85,B 0,C 180,E1 25769.198,E2 25769.198} C_VEL
LIN {X 0,Y 544.343,Z 1007.98,A -85,B 0,C 180,E1 25768.247,E2 25768.247} C_VEL
LIN {X 0,Y 542.405,Z 1028.925,A -85,B 0,C 180,E1 25767.088,E2 25767.088} C_VEL
LIN {X 0,Y 540.401,Z 1048.652,A -85,B 0,C 180,E1 25765.775,E2 25765.775} C_VEL
LIN {X 0,Y 538.38,Z 1067.405,A -85,B 0,C 180,E1 25764.293,E2 25764.293} C_VEL
LIN {X 0,Y 536.397,Z 1084.691,A -85,B 0,C 180,E1 25762.671,E2 25762.671} C_VEL
LIN {X 0,Y 534.675,Z 1099.505,A -85,B 0,C 180,E1 25761.044,E2 25761.044} C_VEL
LIN {X 0,Y 533.094,Z 1113.428,A -85,B 0,C 180,E1 25759.278,E2 25759.278} C_VEL
LIN {X 0,Y 531.63,Z 1126.722,A -85,B 0,C 180,E1 25757.29,E2 25757.29} C_VEL
LIN {X 0,Y 530.468,Z 1137.885,A -85,B 0,C 180,E1 25755.303,E2 25755.303} C_VEL
LIN {X 0,Y 529.524,Z 1148.267,A -85,B 0,C 180,E1 25753.099,E2 25753.099} C_VEL
LIN {X 0,Y 528.866,Z 1156.76,A -85,B 0,C 180,E1 25750.9,E2 25750.9} C_VEL
LIN {X 0,Y 528.438,Z 1163.365,A -85,B 0,C 180,E1 25748.709,E2 25748.709} C_VEL
LIN {X 0,Y 528.18,Z 1168.824,A -85,B 0,C 180,E1 25746.306,E2 25746.306} C_VEL
LIN {X 0,Y 528.062,Z 1172.373,A -85,B 0,C 180,E1 25744.02,E2 25744.02} C_VEL
LIN {X 0,Y 528.022,Z 1174.236,A -85,B 0,C 180,E1 25741.739,E2 25741.739} C_VEL
LIN {X 0,Y 528.013,Z 1174.538,A -85,B 0,C 180,E1 25739.46,E2 25739.46} C_VEL
LIN {X 0,Y 528.025,Z 1173.34,A -85,B 0,C 180,E1 25737.18,E2 25737.18} C_VEL
LIN {X 0,Y 528.078,Z 1170.366,A -85,B 0,C 180,E1 25734.851,E2 25734.851} C_VEL
LIN {X 0,Y 528.227,Z 1165.686,A -85,B 0,C 180,E1 25732.498,E2 25732.498} C_VEL
LIN {X 0,Y 528.526,Z 1159.424,A -85,B 0,C 180,E1 25730.199,E2 25730.199} C_VEL
LIN {X 0,Y 529.005,Z 1151.678,A -85,B 0,C 180,E1 25728.002,E2 25728.002} C_VEL
LIN {X 0,Y 529.686,Z 1142.583,A -85,B 0,C 180,E1 25725.909,E2 25725.909} C_VEL
LIN {X 0,Y 530.665,Z 1131.688,A -85,B 0,C 180,E1 25723.81,E2 25723.81} C_VEL
LIN {X 0,Y 531.89,Z 1119.368,A -85,B 0,C 180,E1 25721.819,E2 25721.819} C_VEL
LIN {X 0,Y 533.336,Z 1105.576,A -85,B 0,C 180,E1 25719.93,E2 25719.93} C_VEL
LIN {X 0,Y 535.088,Z 1089.559,A -85,B 0,C 180,E1 25718.057,E2 25718.057} C_VEL
LIN {X 0,Y 536.923,Z 1072.977,A -85,B 0,C 180,E1 25716.401,E2 25716.401} C_VEL
LIN {X 0,Y 538.819,Z 1055.293,A -85,B 0,C 180,E1 25714.903,E2 25714.903} C_VEL
LIN {X 0,Y 540.744,Z 1036.277,A -85,B 0,C 180,E1 25713.539,E2 25713.539} C_VEL
LIN {X 0,Y 542.619,Z 1016.32,A -85,B 0,C 180,E1 25712.334,E2 25712.334} C_VEL
LIN {X 0,Y 544.369,Z 995.985,A -85,B 0,C 180,E1 25711.315,E2 25711.315} C_VEL
LIN {X 0,Y 545.892,Z 974.72,A -85,B 0,C 180,E1 25710.464,E2 25710.464} C_VEL
LIN {X 0,Y 547.211,Z 952.588,A -85,B 0,C 180,E1 25709.775,E2 25709.775} C_VEL
LIN {X 0,Y 548.241,Z 930.285,A -85,B 0,C 180,E1 25709.268,E2 25709.268} C_VEL
LIN {X 0,Y 555.695,Z 689.445,A -85,B 0,C 180,E1 25705.525,E2 25705.525} C_VEL
LIN {X 0,Y 555.787,Z 683.123,A -85,B 0,C 180,E1 25705.417,E2 25705.417} C_VEL
LIN {X 0,Y 545.03,Z 662.644,A -85,B 0,C 180,E1 25704.34,E2 25704.34} C_VEL
LIN {X 0,Y 531.013,Z 638.215,A -85,B 0,C 180,E1 25702.888,E2 25702.888} C_VEL
LIN {X 0,Y 529.691,Z 634.702,A -85,B 0,C 180,E1 25702.721,E2 25702.721} C_VEL
LIN {X 0,Y 529.688,Z 634.691,A -85,B 0,C 180,E1 25699.225,E2 25699.225} C_VEL
LIN {X 0,Y 529.686,Z 634.689,A -85,B 0,C 180,E1 25695.68,E2 25695.68} C_VEL
LIN {X 0,Y 529.67,Z 634.688,A -85,B 0,C 180,E1 25692.273,E2 25692.273} C_VEL
LIN {X 0,Y 529.609,Z 634.697,A -85,B 0,C 180,E1 25688.941,E2 25688.941} C_VEL
LIN {X 0,Y 529.641,Z 634.688,A -85,B 0,C 180,E1 25685.422,E2 25685.422} C_VEL
LIN {X 0,Y 529.687,Z 634.687,A -85,B 0,C 180,E1 25682.164,E2 25682.164} C_VEL
LIN {X 0,Y 529.686,Z 634.689,A -85,B 0,C 180,E1 25678.862,E2 25678.862} C_VEL
LIN {X 0,Y 528.688,Z 634.817,A -85,B 0,C 180,E1 25678.029,E2 25678.029} C_VEL
LIN {X 0,Y 522.187,Z 635.619,A -85,B 0,C 180,E1 25675.628,E2 25675.628} C_VEL
LIN {X 0,Y 521.722,Z 635.683,A -85,B 0,C 180,E1 25675.079,E2 25675.079} C_VEL
LIN {X 0,Y 521.726,Z 635.677,A -85,B 0,C 180,E1 25671.652,E2 25671.652} C_VEL
LIN {X 0,Y 521.706,Z 635.677,A -85,B 0,C 180,E1 25668.205,E2 25668.205} C_VEL
LIN {X 0,Y 521.719,Z 635.678,A -85,B 0,C 180,E1 25664.769,E2 25664.769} C_VEL
LIN {X 0,Y 521.744,Z 635.674,A -85,B 0,C 180,E1 25661.386,E2 25661.386} C_VEL
LIN {X 0,Y 521.705,Z 635.673,A -85,B 0,C 180,E1 25657.933,E2 25657.933} C_VEL
LIN {X 0,Y 521.684,Z 635.681,A -85,B 0,C 180,E1 25654.509,E2 25654.509} C_VEL
LIN {X 0,Y 521.735,Z 635.678,A -85,B 0,C 180,E1 25650.99,E2 25650.99} C_VEL
LIN {X 0,Y 521.738,Z 635.673,A -85,B 0,C 180,E1 25647.585,E2 25647.585} C_VEL
LIN {X 0,Y 521.743,Z 635.673,A -85,B 0,C 180,E1 25644.062,E2 25644.062} C_VEL
LIN {X 0,Y 521.749,Z 635.673,A -85,B 0,C 180,E1 25640.627,E2 25640.627} C_VEL
LIN {X 0,Y 521.682,Z 635.673,A -85,B 0,C 180,E1 25637.268,E2 25637.268} C_VEL
LIN {X 0,Y 521.675,Z 635.681,A -85,B 0,C 180,E1 25633.751,E2 25633.751} C_VEL
LIN {X 0,Y 521.74,Z 635.674,A -85,B 0,C 180,E1 25630.406,E2 25630.406} C_VEL
LIN {X 0,Y 521.744,Z 635.676,A -85,B 0,C 180,E1 25626.988,E2 25626.988} C_VEL
LIN {X 0,Y 521.738,Z 635.681,A -85,B 0,C 180,E1 25623.481,E2 25623.481} C_VEL
LIN {X 0,Y 521.752,Z 635.679,A -85,B 0,C 180,E1 25620.015,E2 25620.015} C_VEL
LIN {X 0,Y 521.686,Z 635.685,A -85,B 0,C 180,E1 25616.63,E2 25616.63} C_VEL
LIN {X 0,Y 521.703,Z 635.68,A -85,B 0,C 180,E1 25613.233,E2 25613.233} C_VEL
LIN {X 0,Y 521.746,Z 635.675,A -85,B 0,C 180,E1 25609.774,E2 25609.774} C_VEL
LIN {X 0,Y 521.724,Z 635.678,A -85,B 0,C 180,E1 25606.377,E2 25606.377} C_VEL
LIN {X 0,Y 521.738,Z 635.86,A -85,B 0,C 180,E1 25604.216,E2 25604.216} C_VEL
LIN {X 0,Y 529.137,Z 661.681,A -85,B 0,C 180,E1 25601.69,E2 25601.69} C_VEL
LIN {X 0,Y 531.605,Z 671.824,A -85,B 0,C 180,E1 25600.739,E2 25600.739} C_VEL
LIN {X 0,Y 530.288,Z 716.155,A -85,B 0,C 180,E1 25597.152,E2 25597.152} C_VEL
LIN {X 0,Y 528.958,Z 758.88,A -85,B 0,C 180,E1 25593.7,E2 25593.7} C_VEL
LIN {X 0,Y 527.739,Z 799.172,A -85,B 0,C 180,E1 25590.454,E2 25590.454} C_VEL
LIN {X 0,Y 526.818,Z 834.023,A -85,B 0,C 180,E1 25587.693,E2 25587.693} C_VEL
LIN {X 0,Y 526.938,Z 845.258,A -85,B 0,C 180,E1 25587.505,E2 25587.505} C_VEL
LIN {X 0,Y 525.087,Z 977.199,A -85,B 0,C 180,E1 25585.403,E2 25585.403} C_VEL
LIN {X 0,Y 524.91,Z 993.507,A -85,B 0,C 180,E1 25584.95,E2 25584.95} C_VEL
LIN {X 0,Y 524.548,Z 1010.099,A -85,B 0,C 180,E1 25584.275,E2 25584.275} C_VEL
LIN {X 0,Y 524.088,Z 1025.535,A -85,B 0,C 180,E1 25583.416,E2 25583.416} C_VEL
LIN {X 0,Y 523.594,Z 1039.219,A -85,B 0,C 180,E1 25582.446,E2 25582.446} C_VEL
LIN {X 0,Y 523.013,Z 1052.691,A -85,B 0,C 180,E1 25581.237,E2 25581.237} C_VEL
LIN {X 0,Y 522.526,Z 1063.608,A -85,B 0,C 180,E1 25580.028,E2 25580.028} C_VEL
LIN {X 0,Y 522.014,Z 1074.353,A -85,B 0,C 180,E1 25578.537,E2 25578.537} C_VEL
LIN {X 0,Y 521.644,Z 1082.859,A -85,B 0,C 180,E1 25577.051,E2 25577.051} C_VEL
LIN {X 0,Y 521.354,Z 1090.322,A -85,B 0,C 180,E1 25575.344,E2 25575.344} C_VEL
LIN {X 0,Y 521.194,Z 1095.406,A -85,B 0,C 180,E1 25573.759,E2 25573.759} C_VEL
LIN {X 0,Y 521.106,Z 1099.299,A -85,B 0,C 180,E1 25571.893,E2 25571.893} C_VEL
LIN {X 0,Y 521.134,Z 1101.035,A -85,B 0,C 180,E1 25570.164,E2 25570.164} C_VEL
LIN {X 0,Y 521.248,Z 1100.985,A -85,B 0,C 180,E1 25568.38,E2 25568.38} C_VEL
LIN {X 0,Y 521.454,Z 1099.154,A -85,B 0,C 180,E1 25566.674,E2 25566.674} C_VEL
LIN {X 0,Y 521.801,Z 1095.268,A -85,B 0,C 180,E1 25564.867,E2 25564.867} C_VEL
LIN {X 0,Y 522.215,Z 1090.101,A -85,B 0,C 180,E1 25563.291,E2 25563.291} C_VEL
LIN {X 0,Y 522.787,Z 1082.706,A -85,B 0,C 180,E1 25561.642,E2 25561.642} C_VEL
LIN {X 0,Y 523.424,Z 1074.386,A -85,B 0,C 180,E1 25560.217,E2 25560.217} C_VEL
LIN {X 0,Y 524.179,Z 1063.854,A -85,B 0,C 180,E1 25558.795,E2 25558.795} C_VEL
LIN {X 0,Y 524.895,Z 1052.749,A -85,B 0,C 180,E1 25557.596,E2 25557.596} C_VEL
LIN {X 0,Y 525.659,Z 1038.781,A -85,B 0,C 180,E1 25556.399,E2 25556.399} C_VEL
LIN {X 0,Y 526.24,Z 1025.07,A -85,B 0,C 180,E1 25555.475,E2 25555.475} C_VEL
LIN {X 0,Y 526.695,Z 1011.5,A -85,B 0,C 180,E1 25554.769,E2 25554.769} C_VEL
LIN {X 0,Y 527.015,Z 998.635,A -85,B 0,C 180,E1 25554.251,E2 25554.251} C_VEL
LIN {X 0,Y 527.213,Z 983.879,A -85,B 0,C 180,E1 25553.809,E2 25553.809} C_VEL
LIN {X 0,Y 527.633,Z 943.61,A -85,B 0,C 180,E1 25553.109,E2 25553.109} C_VEL
LIN {X 0,Y 530.181,Z 841.855,A -85,B 0,C 180,E1 25551.348,E2 25551.348} C_VEL
LIN {X 0,Y 530.755,Z 833.24,A -85,B 0,C 180,E1 25550.674,E2 25550.674} C_VEL
LIN {X 0,Y 532.235,Z 789.325,A -85,B 0,C 180,E1 25547.19,E2 25547.19} C_VEL
LIN {X 0,Y 533.582,Z 744.397,A -85,B 0,C 180,E1 25543.673,E2 25543.673} C_VEL
LIN {X 0,Y 534.798,Z 701.059,A -85,B 0,C 180,E1 25540.332,E2 25540.332} C_VEL
LIN {X 0,Y 535.427,Z 672.928,A -85,B 0,C 180,E1 25538.182,E2 25538.182} C_VEL
LIN {X 0,Y 530.649,Z 657.45,A -85,B 0,C 180,E1 25536.571,E2 25536.571} C_VEL
LIN {X 0,Y 524.923,Z 643.21,A -85,B 0,C 180,E1 25534.918,E2 25534.918} C_VEL
LIN {X 0,Y 521.92,Z 636.597,A -85,B 0,C 180,E1 25534.098,E2 25534.098} C_VEL
LIN {X 0,Y 521.753,Z 635.681,A -85,B 0,C 180,E1 25533.967,E2 25533.967} C_VEL
LIN {X 0,Y 521.725,Z 635.681,A -85,B 0,C 180,E1 25530.465,E2 25530.465} C_VEL
LIN {X 0,Y 521.722,Z 635.683,A -85,B 0,C 180,E1 25527.153,E2 25527.153} C_VEL
LIN {X 0,Y 521.73,Z 635.679,A -85,B 0,C 180,E1 25523.785,E2 25523.785} C_VEL
LIN {X 0,Y 521.739,Z 635.677,A -85,B 0,C 180,E1 25520.342,E2 25520.342} C_VEL
LIN {X 0,Y 521.74,Z 635.674,A -85,B 0,C 180,E1 25516.677,E2 25516.677} C_VEL
LIN {X 0,Y 521.748,Z 635.675,A -85,B 0,C 180,E1 25513.167,E2 25513.167} C_VEL
LIN {X 0,Y 521.751,Z 635.767,A -85,B 0,C 180,E1 25512.541,E2 25512.541} C_VEL
LIN {X 0,Y 529.893,Z 660.267,A -85,B 0,C 180,E1 25509.144,E2 25509.144} C_VEL
LIN {X 0,Y 535.454,Z 677.637,A -85,B 0,C 180,E1 25506.907,E2 25506.907} C_VEL
LIN {X 0,Y 542.491,Z 692.444,A -85,B 0,C 180,E1 25506.141,E2 25506.141} C_VEL
LIN {X 0,Y 548.839,Z 726.302,A -85,B 0,C 180,E1 25505.097,E2 25505.097} C_VEL
LIN {X 0,Y 541.347,Z 956.64,A -85,B 0,C 180,E1 25501.45,E2 25501.45} C_VEL
LIN {X 0,Y 540.196,Z 987.771,A -85,B 0,C 180,E1 25500.909,E2 25500.909} C_VEL
LIN {X 0,Y 538.869,Z 1010.069,A -85,B 0,C 180,E1 25500.338,E2 25500.338} C_VEL
LIN {X 0,Y 537.235,Z 1032.046,A -85,B 0,C 180,E1 25499.58,E2 25499.58} C_VEL
LIN {X 0,Y 535.397,Z 1053.231,A -85,B 0,C 180,E1 25498.646,E2 25498.646} C_VEL
LIN {X 0,Y 533.421,Z 1073.965,A -85,B 0,C 180,E1 25497.524,E2 25497.524} C_VEL
LIN {X 0,Y 531.387,Z 1093.73,A -85,B 0,C 180,E1 25496.242,E2 25496.242} C_VEL
LIN {X 0,Y 529.358,Z 1112.529,A -85,B 0,C 180,E1 25494.79,E2 25494.79} C_VEL
LIN {X 0,Y 527.444,Z 1129.764,A -85,B 0,C 180,E1 25493.221,E2 25493.221} C_VEL
LIN {X 0,Y 525.534,Z 1147.17,A -85,B 0,C 180,E1 25491.366,E2 25491.366} C_VEL
LIN {X 0,Y 523.975,Z 1162.19,A -85,B 0,C 180,E1 25489.488,E2 25489.488} C_VEL
LIN {X 0,Y 522.644,Z 1175.86,A -85,B 0,C 180,E1 25487.477,E2 25487.477} C_VEL
LIN {X 0,Y 521.601,Z 1187.929,A -85,B 0,C 180,E1 25485.366,E2 25485.366} C_VEL
LIN {X 0,Y 520.829,Z 1198.798,A -85,B 0,C 180,E1 25483.092,E2 25483.092} C_VEL
LIN {X 0,Y 520.368,Z 1207.366,A -85,B 0,C 180,E1 25480.915,E2 25480.915} C_VEL
LIN {X 0,Y 520.112,Z 1214.458,A -85,B 0,C 180,E1 25478.622,E2 25478.622} C_VEL
LIN {X 0,Y 520.005,Z 1219.878,A -85,B 0,C 180,E1 25476.291,E2 25476.291} C_VEL
LIN {X 0,Y 519.994,Z 1223.484,A -85,B 0,C 180,E1 25474.078,E2 25474.078} C_VEL
LIN {X 0,Y 520.011,Z 1225.424,A -85,B 0,C 180,E1 25471.872,E2 25471.872} C_VEL
LIN {X 0,Y 520.01,Z 1225.902,A -85,B 0,C 180,E1 25469.558,E2 25469.558} C_VEL
LIN {X 0,Y 520.006,Z 1224.797,A -85,B 0,C 180,E1 25467.354,E2 25467.354} C_VEL
LIN {X 0,Y 519.99,Z 1221.945,A -85,B 0,C 180,E1 25465.035,E2 25465.035} C_VEL
LIN {X 0,Y 520.038,Z 1217.698,A -85,B 0,C 180,E1 25462.814,E2 25462.814} C_VEL
LIN {X 0,Y 520.169,Z 1211.73,A -85,B 0,C 180,E1 25460.595,E2 25460.595} C_VEL
LIN {X 0,Y 520.498,Z 1203.599,A -85,B 0,C 180,E1 25458.249,E2 25458.249} C_VEL
LIN {X 0,Y 521.033,Z 1194.499,A -85,B 0,C 180,E1 25456.119,E2 25456.119} C_VEL
LIN {X 0,Y 521.836,Z 1183.409,A -85,B 0,C 180,E1 25453.982,E2 25453.982} C_VEL
LIN {X 0,Y 522.95,Z 1170.306,A -85,B 0,C 180,E1 25451.859,E2 25451.859} C_VEL
LIN {X 0,Y 524.304,Z 1156.252,A -85,B 0,C 180,E1 25449.922,E2 25449.922} C_VEL
LIN {X 0,Y 525.9,Z 1140.837,A -85,B 0,C 180,E1 25448.102,E2 25448.102} C_VEL
LIN {X 0,Y 527.65,Z 1124.268,A -85,B 0,C 180,E1 25446.43,E2 25446.43} C_VEL
LIN {X 0,Y 529.675,Z 1105.484,A -85,B 0,C 180,E1 25444.805,E2 25444.805} C_VEL
LIN {X 0,Y 531.798,Z 1085.776,A -85,B 0,C 180,E1 25443.356,E2 25443.356} C_VEL
LIN {X 0,Y 533.915,Z 1065.223,A -85,B 0,C 180,E1 25442.082,E2 25442.082} C_VEL
LIN {X 0,Y 535.994,Z 1043.781,A -85,B 0,C 180,E1 25440.985,E2 25440.985} C_VEL
LIN {X 0,Y 538.033,Z 1021.016,A -85,B 0,C 180,E1 25440.035,E2 25440.035} C_VEL
LIN {X 0,Y 540.025,Z 996.55,A -85,B 0,C 180,E1 25439.242,E2 25439.242} C_VEL
LIN {X 0,Y 541.647,Z 972.483,A -85,B 0,C 180,E1 25438.667,E2 25438.667} C_VEL
LIN {X 0,Y 546.564,Z 874.605,A -85,B 0,C 180,E1 25436.818,E2 25436.818} C_VEL
LIN {X 0,Y 552.524,Z 788.983,A -85,B 0,C 180,E1 25435.06,E2 25435.06} C_VEL
LIN {X 0,Y 557.926,Z 726.427,A -85,B 0,C 180,E1 25433.689,E2 25433.689} C_VEL
LIN {X 0,Y 556.383,Z 705.28,A -85,B 0,C 180,E1 25432.699,E2 25432.699} C_VEL
LIN {X 0,Y 555.757,Z 700.714,A -85,B 0,C 180,E1 25432.424,E2 25432.424} C_VEL
LIN {X 0,Y 552.004,Z 691.407,A -85,B 0,C 180,E1 25431.389,E2 25431.389} C_VEL
LIN {X 0,Y 548.06,Z 682.955,A -85,B 0,C 180,E1 25430.143,E2 25430.143} C_VEL
LIN {X 0,Y 544.278,Z 675.432,A -85,B 0,C 180,E1 25428.624,E2 25428.624} C_VEL
LIN {X 0,Y 542.23,Z 671.809,A -85,B 0,C 180,E1 25427.53,E2 25427.53} C_VEL
LIN {X 0,Y 541.095,Z 669.48,A -85,B 0,C 180,E1 25426.65,E2 25426.65} C_VEL
LIN {X 0,Y 540.092,Z 666.661,A -85,B 0,C 180,E1 25424.991,E2 25424.991} C_VEL
LIN {X 0,Y 540.569,Z 666.372,A -85,B 0,C 180,E1 25423.369,E2 25423.369} C_VEL
LIN {X 0,Y 541.987,Z 667.104,A -85,B 0,C 180,E1 25422.128,E2 25422.128} C_VEL
LIN {X 0,Y 544.033,Z 669.435,A -85,B 0,C 180,E1 25420.94,E2 25420.94} C_VEL
LIN {X 0,Y 547.963,Z 674.045,A -85,B 0,C 180,E1 25419.395,E2 25419.395} C_VEL
LIN {X 0,Y 551.977,Z 680,A -85,B 0,C 180,E1 25418.169,E2 25418.169} C_VEL
LIN {X 0,Y 555.968,Z 686.268,A -85,B 0,C 180,E1 25417.16,E2 25417.16} C_VEL
LIN {X 0,Y 560.204,Z 694.199,A -85,B 0,C 180,E1 25416.19,E2 25416.19} C_VEL
LIN {X 0,Y 552.347,Z 778.477,A -85,B 0,C 180,E1 25414.349,E2 25414.349} C_VEL
LIN {X 0,Y 546.777,Z 857.147,A -85,B 0,C 180,E1 25412.736,E2 25412.736} C_VEL
LIN {X 0,Y 542.226,Z 943.303,A -85,B 0,C 180,E1 25411.062,E2 25411.062} C_VEL
LIN {X 0,Y 540.834,Z 966.338,A -85,B 0,C 180,E1 25410.414,E2 25410.414} C_VEL
LIN {X 0,Y 539.153,Z 988.471,A -85,B 0,C 180,E1 25409.596,E2 25409.596} C_VEL
LIN {X 0,Y 537.296,Z 1009.53,A -85,B 0,C 180,E1 25408.616,E2 25408.616} C_VEL
LIN {X 0,Y 535.289,Z 1029.848,A -85,B 0,C 180,E1 25407.466,E2 25407.466} C_VEL
LIN {X 0,Y 533.195,Z 1049.294,A -85,B 0,C 180,E1 25406.15,E2 25406.15} C_VEL
LIN {X 0,Y 531.063,Z 1067.984,A -85,B 0,C 180,E1 25404.65,E2 25404.65} C_VEL
LIN {X 0,Y 528.94,Z 1085.475,A -85,B 0,C 180,E1 25402.983,E2 25402.983} C_VEL
LIN {X 0,Y 527.034,Z 1100.955,A -85,B 0,C 180,E1 25401.248,E2 25401.248} C_VEL
LIN {X 0,Y 525.277,Z 1115.473,A -85,B 0,C 180,E1 25399.345,E2 25399.345} C_VEL
LIN {X 0,Y 523.843,Z 1127.914,A -85,B 0,C 180,E1 25397.44,E2 25397.44} C_VEL
LIN {X 0,Y 522.558,Z 1139.52,A -85,B 0,C 180,E1 25395.313,E2 25395.313} C_VEL
LIN {X 0,Y 521.579,Z 1149.661,A -85,B 0,C 180,E1 25393.076,E2 25393.076} C_VEL
LIN {X 0,Y 520.899,Z 1157.937,A -85,B 0,C 180,E1 25390.845,E2 25390.845} C_VEL
LIN {X 0,Y 520.465,Z 1164.434,A -85,B 0,C 180,E1 25388.62,E2 25388.62} C_VEL
LIN {X 0,Y 520.202,Z 1169.482,A -85,B 0,C 180,E1 25386.292,E2 25386.292} C_VEL
LIN {X 0,Y 520.075,Z 1172.919,A -85,B 0,C 180,E1 25383.971,E2 25383.971} C_VEL
LIN {X 0,Y 520.033,Z 1174.661,A -85,B 0,C 180,E1 25381.765,E2 25381.765} C_VEL
LIN {X 0,Y 520.023,Z 1174.934,A -85,B 0,C 180,E1 25379.452,E2 25379.452} C_VEL
LIN {X 0,Y 520.036,Z 1173.694,A -85,B 0,C 180,E1 25377.137,E2 25377.137} C_VEL
LIN {X 0,Y 520.092,Z 1170.724,A -85,B 0,C 180,E1 25374.795,E2 25374.795} C_VEL
LIN {X 0,Y 520.252,Z 1165.947,A -85,B 0,C 180,E1 25372.382,E2 25372.382} C_VEL
LIN {X 0,Y 520.553,Z 1159.975,A -85,B 0,C 180,E1 25370.159,E2 25370.159} C_VEL
LIN {X 0,Y 521.05,Z 1152.229,A -85,B 0,C 180,E1 25367.929,E2 25367.929} C_VEL
LIN {X 0,Y 521.808,Z 1142.626,A -85,B 0,C 180,E1 25365.691,E2 25365.691} C_VEL
LIN {X 0,Y 522.839,Z 1131.629,A -85,B 0,C 180,E1 25363.561,E2 25363.561} C_VEL
LIN {X 0,Y 524.202,Z 1118.608,A -85,B 0,C 180,E1 25361.444,E2 25361.444} C_VEL
LIN {X 0,Y 525.742,Z 1104.495,A -85,B 0,C 180,E1 25359.519,E2 25359.519} C_VEL
LIN {X 0,Y 527.487,Z 1089.122,A -85,B 0,C 180,E1 25357.724,E2 25357.724} C_VEL
LIN {X 0,Y 529.395,Z 1072.339,A -85,B 0,C 180,E1 25356.044,E2 25356.044} C_VEL
LIN {X 0,Y 531.455,Z 1053.964,A -85,B 0,C 180,E1 25354.482,E2 25354.482} C_VEL
LIN {X 0,Y 533.389,Z 1035.275,A -85,B 0,C 180,E1 25353.145,E2 25353.145} C_VEL
LIN {X 0,Y 535.353,Z 1015.02,A -85,B 0,C 180,E1 25351.926,E2 25351.926} C_VEL
LIN {X 0,Y 537.093,Z 995.175,A -85,B 0,C 180,E1 25350.932,E2 25350.932} C_VEL
LIN {X 0,Y 538.667,Z 974.047,A -85,B 0,C 180,E1 25350.082,E2 25350.082} C_VEL
LIN {X 0,Y 540.006,Z 952.215,A -85,B 0,C 180,E1 25349.401,E2 25349.401} C_VEL
LIN {X 0,Y 541.084,Z 928.923,A -85,B 0,C 180,E1 25348.875,E2 25348.875} C_VEL
LIN {X 0,Y 549.013,Z 685.94,A -85,B 0,C 180,E1 25345.031,E2 25345.031} C_VEL
LIN {X 0,Y 538.955,Z 666.926,A -85,B 0,C 180,E1 25344.011,E2 25344.011} C_VEL
LIN {X 0,Y 523.192,Z 639.375,A -85,B 0,C 180,E1 25342.345,E2 25342.345} C_VEL
LIN {X 0,Y 521.779,Z 636.034,A -85,B 0,C 180,E1 25342.173,E2 25342.173} C_VEL
LIN {X 0,Y 521.724,Z 635.676,A -85,B 0,C 180,E1 25342.15,E2 25342.15} C_VEL
LIN {X 0,Y 521.745,Z 635.674,A -85,B 0,C 180,E1 25338.761,E2 25338.761} C_VEL
LIN {X 0,Y 521.728,Z 635.681,A -85,B 0,C 180,E1 25335.308,E2 25335.308} C_VEL
LIN {X 0,Y 521.746,Z 635.677,A -85,B 0,C 180,E1 25331.968,E2 25331.968} C_VEL
LIN {X 0,Y 521.69,Z 635.686,A -85,B 0,C 180,E1 25328.562,E2 25328.562} C_VEL
LIN {X 0,Y 521.699,Z 635.678,A -85,B 0,C 180,E1 25325.234,E2 25325.234} C_VEL
LIN {X 0,Y 521.745,Z 635.674,A -85,B 0,C 180,E1 25321.805,E2 25321.805} C_VEL
LIN {X 0,Y 521.728,Z 635.68,A -85,B 0,C 180,E1 25318.379,E2 25318.379} C_VEL
LIN {X 0,Y 521.722,Z 635.683,A -85,B 0,C 180,E1 25315.079,E2 25315.079} C_VEL
LIN {X 0,Y 520.706,Z 635.818,A -85,B 0,C 180,E1 25314.234,E2 25314.234} C_VEL
LIN {X 0,Y 514.225,Z 636.615,A -85,B 0,C 180,E1 25311.796,E2 25311.796} C_VEL
LIN {X 0,Y 513.757,Z 636.674,A -85,B 0,C 180,E1 25311.238,E2 25311.238} C_VEL
LIN {X 0,Y 513.803,Z 636.662,A -85,B 0,C 180,E1 25307.791,E2 25307.791} C_VEL
LIN {X 0,Y 513.802,Z 636.662,A -85,B 0,C 180,E1 25304.286,E2 25304.286} C_VEL
LIN {X 0,Y 513.805,Z 636.667,A -85,B 0,C 180,E1 25300.769,E2 25300.769} C_VEL
LIN {X 0,Y 513.787,Z 636.66,A -85,B 0,C 180,E1 25297.381,E2 25297.381} C_VEL
LIN {X 0,Y 513.727,Z 636.67,A -85,B 0,C 180,E1 25294.019,E2 25294.019} C_VEL
LIN {X 0,Y 513.755,Z 636.669,A -85,B 0,C 180,E1 25290.448,E2 25290.448} C_VEL
LIN {X 0,Y 513.808,Z 636.654,A -85,B 0,C 180,E1 25287.101,E2 25287.101} C_VEL
LIN {X 0,Y 513.798,Z 636.668,A -85,B 0,C 180,E1 25283.633,E2 25283.633} C_VEL
LIN {X 0,Y 513.795,Z 636.658,A -85,B 0,C 180,E1 25280.141,E2 25280.141} C_VEL
LIN {X 0,Y 513.794,Z 636.662,A -85,B 0,C 180,E1 25276.611,E2 25276.611} C_VEL
LIN {X 0,Y 513.759,Z 636.671,A -85,B 0,C 180,E1 25273.145,E2 25273.145} C_VEL
LIN {X 0,Y 513.776,Z 636.666,A -85,B 0,C 180,E1 25269.716,E2 25269.716} C_VEL
LIN {X 0,Y 513.809,Z 636.661,A -85,B 0,C 180,E1 25266.247,E2 25266.247} C_VEL
LIN {X 0,Y 513.776,Z 636.667,A -85,B 0,C 180,E1 25262.786,E2 25262.786} C_VEL
LIN {X 0,Y 513.746,Z 636.673,A -85,B 0,C 180,E1 25259.338,E2 25259.338} C_VEL
LIN {X 0,Y 513.78,Z 636.672,A -85,B 0,C 180,E1 25255.913,E2 25255.913} C_VEL
LIN {X 0,Y 513.802,Z 636.67,A -85,B 0,C 180,E1 25252.477,E2 25252.477} C_VEL
